// Exactly 1 after an abandon, however many scans the runner has left.
PROPERTY AbandonCalls : UDINT
GET
AbandonCalls := _AbandonCalls;
END_GET
END_PROPERTY

PROPERTY BodyCalls : UDINT
GET
BodyCalls := _BodyCalls;
END_GET
END_PROPERTY

METHOD Run : BOOL
VAR_INPUT
	Enable : BOOL;
	Test   : I_TestAssertions;
END_VAR
IF NOT Enable THEN
	_AbandonCalls := _AbandonCalls + 1;

	// Deliberately does NOT report itself finished. A test that hung will not

	// answer this either, and the runner must not wait for it.
	Run := FALSE;
	RETURN;
END_IF

_BodyCalls := _BodyCalls + 1;
Run		   := FALSE;
END_METHOD

// Always 0 - this double implements no teardown. Declared so a test can assert

// that abandonment did not somehow invent one.
PROPERTY TeardownCalls : UDINT
GET
TeardownCalls := 0;
END_GET
END_PROPERTY

END_FUNCTION_BLOCK

// ---- Tests/Runner/TEST_RunnerSetupDeadlineFires.TcPOU
// Setup has its OWN deadline. A fixture that never comes up must not run forever

// on the body's budget, and the body must never be reached.

//

// Teardown still runs: a fixture that half came up is exactly when cleanup

// matters.
FUNCTION_BLOCK TEST_RunnerSetupDeadlineFires IMPLEMENTS I_Test
VAR
	// A private runner, driven one scan per call. The outer test spans scans by

	// returning FALSE, which is exactly the mechanism being verified one level down.
	Registry	 : TestRegistry<1>;
	Runner		 : TestRunner;
	Handle		 : TestVerdict;
	Budgets		 : ST_TestBudgets;
	Journal		 : REFERENCE TO TestJournal;
	Slot		 : ST_TestSlot;
	Outcome		 : E_PhaseOutcome;
	Loaded		 : BOOL;
	Phase		 : DINT;
	Scans		 : DINT;
	Subject		 : HangingSetupTest;
	ExpectedZero : UDINT;
	ExpectedOne	 : UDINT;
	ExpectedTwo	 : UDINT;
	ActualCount	 : UDINT;
	ExpectedKind : E_FailureKind;
	ActualKind	 : E_FailureKind;
END_VAR

METHOD Run : BOOL
VAR_INPUT
	Enable : BOOL;
	Test   : I_TestAssertions;
END_VAR
Scans := Scans + 1;
IF Scans > 200 THEN
	Test.Fail('the subject never reached a terminal outcome');
	Run := TRUE;
	RETURN;
END_IF

CASE Phase OF
	0:
		Budgets.Setup.Cycles	  := 2;
		Budgets.Setup.IsCyclesSet := TRUE;

		// The body budget is deliberately left disabled. If the runner were using it

		// for setup, nothing would ever expire and the watchdog would fail this test.
		Registry.TryClaim(Subject, 'setup hangs', Budgets);
		Runner.Attach(Roster := Registry, Verdict := Handle);
		Slot   := Registry.Slot(0);
		Loaded := Runner.Load(Slot);
		Phase  := 1;
		Run	   := FALSE;

	1:
		Outcome := Runner.Advance(Enable := TRUE);
		IF Outcome <> E_PhaseOutcome.Running THEN
			Phase := 2;
		END_IF

		Run := FALSE;

	2:
		ExpectedTwo := 2;
		ActualCount := Subject.SetupCalls;
		Test.AssertEqual(ExpectedTwo, ActualCount, 'setup got its own budget, not the body one');
		ExpectedZero := 0;
		ActualCount	 := Subject.BodyCalls;
		Test.AssertEqual(ExpectedZero, ActualCount, 'the body was never reached');
		ExpectedOne := 1;
		ActualCount := Subject.TeardownCalls;
		Test.AssertEqual(ExpectedOne, ActualCount, 'teardown ran anyway');
		Journal REF= Registry.Journal(0);
		IF __ISVALIDREF(Journal) THEN
			ExpectedKind := E_FailureKind.Timeout;
			ActualKind	 := Journal.Kind;
			Test.AssertEqual(ExpectedKind, ActualKind, 'recorded as a timeout');
		END_IF

		Run := TRUE;
END_CASE
END_METHOD

END_FUNCTION_BLOCK

// ---- Doubles/HangingSetupTest.TcPOU
// Setup that never completes. Bounded by the SETUP deadline, not the body's - the

// body must never run, and teardown must still be called.
FUNCTION_BLOCK HangingSetupTest IMPLEMENTS I_Test, I_TestSetup, I_TestTeardown
VAR
	_SetupCalls	   : UDINT;
	_BodyCalls	   : UDINT;
	_TeardownCalls : UDINT;
END_VAR

// Must be 0. Setup never succeeded, so the body was never exercised.
PROPERTY BodyCalls : UDINT
GET
BodyCalls := _BodyCalls;
END_GET
END_PROPERTY

METHOD Run : BOOL
VAR_INPUT
	Enable : BOOL;
	Test   : I_TestAssertions;
END_VAR
IF Enable THEN
	_BodyCalls := _BodyCalls + 1;
END_IF

Run := TRUE;
END_METHOD

METHOD Setup : BOOL
VAR_INPUT
	Enable : BOOL;
	Test   : I_TestAssertions;
END_VAR
IF Enable THEN
	_SetupCalls := _SetupCalls + 1;
END_IF

Setup := FALSE;
END_METHOD

PROPERTY SetupCalls : UDINT
GET
SetupCalls := _SetupCalls;
END_GET
END_PROPERTY

METHOD Teardown : BOOL
VAR_INPUT
	Enable : BOOL;
	Test   : I_TestAssertions;
END_VAR
_TeardownCalls := _TeardownCalls + 1;
Teardown	   := TRUE;
END_METHOD

// Must be 1 even here. On a rig, a fixture that half came up is exactly when

// cleanup matters most.
PROPERTY TeardownCalls : UDINT
GET
TeardownCalls := _TeardownCalls;
END_GET
END_PROPERTY

END_FUNCTION_BLOCK

// ---- Tests/Runner/TEST_RunnerTeardownOverrunKeepsTheVerdict.TcPOU
// A passing test whose cleanup hangs still proved the code correct. The verdict

// stands.

//

// The overrun is reported separately - TeardownOverran, with a diagnostic and the

// label - because the SUITE has to raise a framework error for it and the runner

// holds no reporters. On a rig this may mean an axis left powered, so it must be

// loud without being a lie about the test.
FUNCTION_BLOCK TEST_RunnerTeardownOverrunKeepsTheVerdict IMPLEMENTS I_Test
VAR
	// A private runner, driven one scan per call. The outer test spans scans by

	// returning FALSE, which is exactly the mechanism being verified one level down.
	Registry	   : TestRegistry<1>;
	Runner		   : TestRunner;
	Handle		   : TestVerdict;
	Budgets		   : ST_TestBudgets;
	Journal		   : REFERENCE TO TestJournal;
	Slot		   : ST_TestSlot;
	Outcome		   : E_PhaseOutcome;
	Loaded		   : BOOL;
	Phase		   : DINT;
	Scans		   : DINT;
	Subject		   : HangingTeardownTest;
	ExpectedTwo	   : UDINT;
	ActualCount	   : UDINT;
	ExpectedStatus : E_TestStatus;
	ActualStatus   : E_TestStatus;
	Diagnostic	   : T_MaxString;
	ActiveLabel	   : T_MaxString;
	ExpectedLabel  : T_MaxString;
END_VAR

METHOD Run : BOOL
VAR_INPUT
	Enable : BOOL;
	Test   : I_TestAssertions;
END_VAR
Scans := Scans + 1;
IF Scans > 200 THEN
	Test.Fail('the subject never reached a terminal outcome');
	Run := TRUE;
	RETURN;
END_IF

CASE Phase OF
	0:
		Budgets.Teardown.Cycles		 := 2;
		Budgets.Teardown.IsCyclesSet := TRUE;
		Registry.TryClaim(Subject, 'teardown hangs', Budgets);
		Runner.Attach(Roster := Registry, Verdict := Handle);
		Slot   := Registry.Slot(0);
		Loaded := Runner.Load(Slot);
		Phase  := 1;
		Run	   := FALSE;

	1:
		Outcome := Runner.Advance(Enable := TRUE);
		IF Outcome <> E_PhaseOutcome.Running THEN
			// Read before anything else can unload it.
			Diagnostic	:= Runner.TeardownDiagnostic;
			ActiveLabel := Runner.ActiveLabel;
			Phase		:= 2;
		END_IF

		Run := FALSE;

	2:
		Test.AssertTrue(Outcome = E_PhaseOutcome.TeardownOverran, 'reported as an overrun');
		ExpectedTwo := 2;
		ActualCount := Subject.TeardownCalls;
		Test.AssertEqual(ExpectedTwo, ActualCount, 'teardown got its own budget');
		Test.AssertTrue(Diagnostic <> '', 'a diagnostic was composed');
		Test.AssertTrue(FIND(Diagnostic, 'teardown') > 0, 'and it names the phase');
		ExpectedLabel := 'teardown hangs';
		Test.AssertEqual(ExpectedLabel, ActiveLabel, 'and the test that hung');

		// The point of the whole test.
		Journal REF= Registry.Journal(0);
		IF __ISVALIDREF(Journal) THEN
			ExpectedStatus := E_TestStatus.Passed;
			ActualStatus   := Journal.Status;
			Test.AssertEqual(ExpectedStatus, ActualStatus, 'the verdict is untouched');
		END_IF

		Run := TRUE;
END_CASE
END_METHOD

END_FUNCTION_BLOCK

// ---- Doubles/HangingTeardownTest.TcPOU
// Passes cleanly, then hangs on the way out.

//

// The verdict must survive: a passing test whose cleanup hung still proved the

// code correct. The overrun is a framework error, not a test failure - but on a

// rig it may mean an axis left powered, so it must be loud.
FUNCTION_BLOCK HangingTeardownTest IMPLEMENTS I_Test, I_TestTeardown
VAR
	_BodyCalls	   : UDINT;
	_TeardownCalls : UDINT;
END_VAR

PROPERTY BodyCalls : UDINT
GET
BodyCalls := _BodyCalls;
END_GET
END_PROPERTY

METHOD Run : BOOL
VAR_INPUT
	Enable : BOOL;
	Test   : I_TestAssertions;
END_VAR
IF Enable THEN
	_BodyCalls := _BodyCalls + 1;
	Test.AssertTrue(TRUE, 'the body was fine');
END_IF

Run := TRUE;
END_METHOD

METHOD Teardown : BOOL
VAR_INPUT
	Enable : BOOL;
	Test   : I_TestAssertions;
END_VAR
IF Enable THEN
	_TeardownCalls := _TeardownCalls + 1;
END_IF

Teardown := FALSE;
END_METHOD

PROPERTY TeardownCalls : UDINT
GET
TeardownCalls := _TeardownCalls;
END_GET
END_PROPERTY

END_FUNCTION_BLOCK

// ---- Tests/Runner/TEST_RunnerAbandonMakesOneFinalCall.TcPOU
// Dropping Enable abandons the test. The phase in flight gets ONE final call so

// it can put its own state back, and the return is ignored - a test that hung will

// not answer that call either, and waiting for it would reproduce the stall the

// design removes.

//

// Teardown is NOT run. Abandonment is the suite being switched off, not a test

// finishing, and calling cleanup on a half-torn-down rig is its own hazard.
FUNCTION_BLOCK TEST_RunnerAbandonMakesOneFinalCall IMPLEMENTS I_Test
VAR
	// A private runner, driven one scan per call. The outer test spans scans by

	// returning FALSE, which is exactly the mechanism being verified one level down.
	Registry	   : TestRegistry<1>;
	Runner		   : TestRunner;
	Handle		   : TestVerdict;
	Budgets		   : ST_TestBudgets;
	Journal		   : REFERENCE TO TestJournal;
	Slot		   : ST_TestSlot;
	Outcome		   : E_PhaseOutcome;
	Loaded		   : BOOL;
	Phase		   : DINT;
	Scans		   : DINT;
	Subject		   : HangingBodyTest;
	ExpectedOne	   : UDINT;
	ExpectedZero   : UDINT;
	ActualCount	   : UDINT;
	ExpectedStatus : E_TestStatus;
	ActualStatus   : E_TestStatus;
END_VAR

METHOD Run : BOOL
VAR_INPUT
	Enable : BOOL;
	Test   : I_TestAssertions;
END_VAR
Scans := Scans + 1;
IF Scans > 200 THEN
	Test.Fail('the subject never reached a terminal outcome');
	Run := TRUE;
	RETURN;
END_IF

CASE Phase OF
	0:
		Registry.TryClaim(Subject, 'abandoned', Budgets);
		Runner.Attach(Roster := Registry, Verdict := Handle);
		Slot   := Registry.Slot(0);
		Loaded := Runner.Load(Slot);
		Phase  := 1;
		Run	   := FALSE;

	1:
		// Let it run a couple of scans first, so there is something to abandon.
		Outcome := Runner.Advance(Enable := TRUE);
		IF Subject.BodyCalls >= 2 THEN
			Phase := 2;
		END_IF

		Run := FALSE;

	2:
		Outcome := Runner.Advance(Enable := FALSE);
		Phase	:= 3;
		Run		:= FALSE;

	3:
		// A second abandon must not produce a second final call.
		Outcome := Runner.Advance(Enable := FALSE);
		Phase	:= 4;
		Run		:= FALSE;

	4:
		ExpectedOne := 1;
		ActualCount := Subject.AbandonCalls;
		Test.AssertEqual(ExpectedOne, ActualCount, 'exactly one call with Enable FALSE');
		ExpectedZero := 0;
		ActualCount	 := Subject.TeardownCalls;
		Test.AssertEqual(ExpectedZero, ActualCount, 'teardown was not run');
		Journal REF= Registry.Journal(0);
		IF __ISVALIDREF(Journal) THEN
			// Errored, not Failed: the code under test was never shown to be wrong. Not
			// Skipped either - an abandoned run must not read as a clean one.
			ExpectedStatus := E_TestStatus.Errored;
			ActualStatus   := Journal.Status;
			Test.AssertEqual(ExpectedStatus, ActualStatus, 'abandoned tests are Errored');
		END_IF

		Run := TRUE;
END_CASE
END_METHOD

END_FUNCTION_BLOCK

// ---- Tests/Runner/TEST_RunnerRefusesAnEmptySlot.TcPOU
// A slot carrying no test is refused, and nothing is loaded. A caller that has

// miscounted gets FALSE and an Idle runner rather than a dereferenced null.
FUNCTION_BLOCK TEST_RunnerRefusesAnEmptySlot IMPLEMENTS I_Test
VAR
	// A private runner, driven one scan per call. The outer test spans scans by

	// returning FALSE, which is exactly the mechanism being verified one level down.
	Registry  : TestRegistry<1>;
	Runner	  : TestRunner;
	Handle	  : TestVerdict;
	Budgets	  : ST_TestBudgets;
	Journal	  : REFERENCE TO TestJournal;
	Slot	  : ST_TestSlot;
	Outcome	  : E_PhaseOutcome;
	Loaded	  : BOOL;
	Phase	  : DINT;
	Scans	  : DINT;
	EmptySlot : ST_TestSlot;
	Refused	  : BOOL;
END_VAR

METHOD Run : BOOL
VAR_INPUT
	Enable : BOOL;
	Test   : I_TestAssertions;
END_VAR
Scans := Scans + 1;
IF Scans > 200 THEN
	Test.Fail('the subject never reached a terminal outcome');
	Run := TRUE;
	RETURN;
END_IF

Runner.Attach(Roster := Registry, Verdict := Handle);
Refused := Runner.Load(EmptySlot);
Test.AssertFalse(Refused, 'an empty slot is refused');
Test.AssertTrue(Runner.Outcome = E_PhaseOutcome.Idle, 'and nothing was loaded');

// Slot 0 of an empty registry is also empty - the registry hands back a defined

// empty slot rather than whatever was nearby.
Slot	:= Registry.Slot(0);
Refused := Runner.Load(Slot);
Test.AssertFalse(Refused, 'an unregistered index is refused too');
Test.AssertTrue(Runner.Outcome = E_PhaseOutcome.Idle, 'still nothing loaded');
Run := TRUE;
END_METHOD

END_FUNCTION_BLOCK

// ---- Tests/Suite/TEST_SuiteRunsEveryRegisteredTest.TcPOU
// The whole loop: register three, drive to completion, and every one of them ran

// exactly once and was counted.
FUNCTION_BLOCK TEST_SuiteRunsEveryRegisteredTest IMPLEMENTS I_Test
VAR
	// A private suite, driven one scan per call. The outer test spans scans by

	// returning FALSE - which is the mechanism the inner suite is being asked to

	// drive, one level down.
	Inner			: TestSuite<4>;
	Budgets			: ST_TestBudgets;
	Phase			: DINT;
	Scans			: DINT;
	A				: PassingTest;
	B				: PassingTest;
	C				: PassingTest;
	ExpectedCount	: UDINT;
	ActualCount		: UDINT;
	ExpectedOutcome : E_RunOutcome;
	ActualOutcome	: E_RunOutcome;
END_VAR

METHOD Run : BOOL
VAR_INPUT
	Enable : BOOL;
	Test   : I_TestAssertions;
END_VAR
Scans := Scans + 1;
IF Scans > 200 THEN
	Test.Fail('the inner suite never completed');
	Run := TRUE;
	RETURN;
END_IF

CASE Phase OF
	0:
		Inner.SetLabel('inner');
		Inner.Register(A, 'first', Budgets);
		Inner.Register(B, 'second', Budgets);
		Inner.Register(C, 'third', Budgets);
		Phase := 1;
		Run	  := FALSE;

	1:
		IF Inner.Run(Enable := TRUE) THEN
			Phase := 2;
		END_IF

		Run := FALSE;

	2:
		Test.AssertTrue(Inner.IsComplete, 'the run finished');
		ExpectedCount := 3;
		ActualCount	  := Inner.TestCount;
		Test.AssertEqual(ExpectedCount, ActualCount, 'three registered');
		ActualCount := Inner.PassedCount;
		Test.AssertEqual(ExpectedCount, ActualCount, 'three passed');
		ExpectedCount := 0;
		ActualCount	  := Inner.FailedCount;
		Test.AssertEqual(ExpectedCount, ActualCount, 'none failed');
		ExpectedCount := 1;
		ActualCount	  := A.BodyCalls;
		Test.AssertEqual(ExpectedCount, ActualCount, 'the first ran once');
		ActualCount := C.BodyCalls;
		Test.AssertEqual(ExpectedCount, ActualCount, 'and so did the last');
		ExpectedOutcome := E_RunOutcome.Passed;
		ActualOutcome	:= Inner.Outcome;
		Test.AssertEqual(ExpectedOutcome, ActualOutcome, 'the run passed');
		Run := TRUE;
END_CASE
END_METHOD

END_FUNCTION_BLOCK

// ---- Doubles/PassingTest.TcPOU
// Passes in one scan. The baseline for suite-level counting.

//

// Records a check deliberately: a body that checks nothing is reported Errored,

// not Passed, so a double that asserted nothing would quietly test the wrong

// thing.
FUNCTION_BLOCK PassingTest IMPLEMENTS I_Test
VAR
	_BodyCalls : UDINT;
END_VAR

// How many times a suite has run this. A re-run doubles it; an individual re-run

// raises it without touching any count the suite reports.
PROPERTY BodyCalls : UDINT
GET
BodyCalls := _BodyCalls;
END_GET
END_PROPERTY

METHOD Run : BOOL
VAR_INPUT
	Enable : BOOL;
	Test   : I_TestAssertions;
END_VAR
IF NOT Enable THEN
	Run := TRUE;
	RETURN;
END_IF

_BodyCalls := _BodyCalls + 1;
Test.AssertTrue(TRUE, 'this one passes');
Run := TRUE;
END_METHOD

END_FUNCTION_BLOCK

// ---- Tests/Suite/TEST_SuiteSeparatesFailuresFromErrors.TcPOU
// Failed and Errored are different signals and are counted apart.

//

// A failure means the code is wrong. An error means the run cannot be trusted -

// and Errored outranks Failed in the aggregate, because a framework or environment

// problem casts doubt on every other result.
FUNCTION_BLOCK TEST_SuiteSeparatesFailuresFromErrors IMPLEMENTS I_Test
VAR
	// A private suite, driven one scan per call. The outer test spans scans by

	// returning FALSE - which is the mechanism the inner suite is being asked to

	// drive, one level down.
	Inner			: TestSuite<4>;
	Budgets			: ST_TestBudgets;
	Phase			: DINT;
	Scans			: DINT;
	Good			: PassingTest;
	Bad				: FailingTest;
	Ugly			: ErroringTest;
	ExpectedCount	: UDINT;
	ActualCount		: UDINT;
	ExpectedOutcome : E_RunOutcome;
	ActualOutcome	: E_RunOutcome;
END_VAR

METHOD Run : BOOL
VAR_INPUT
	Enable : BOOL;
	Test   : I_TestAssertions;
END_VAR
Scans := Scans + 1;
IF Scans > 200 THEN
	Test.Fail('the inner suite never completed');
	Run := TRUE;
	RETURN;
END_IF

CASE Phase OF
	0:
		Inner.SetLabel('inner');
		Inner.Register(Good, 'passes', Budgets);
		Inner.Register(Bad, 'fails', Budgets);
		Inner.Register(Ugly, 'errors', Budgets);
		Phase := 1;
		Run	  := FALSE;

	1:
		IF Inner.Run(Enable := TRUE) THEN
			Phase := 2;
		END_IF

		Run := FALSE;

	2:
		ExpectedCount := 1;
		ActualCount	  := Inner.PassedCount;
		Test.AssertEqual(ExpectedCount, ActualCount, 'one passed');
		ActualCount := Inner.FailedCount;
		Test.AssertEqual(ExpectedCount, ActualCount, 'one failed');
		ActualCount := Inner.ErrorCount;
		Test.AssertEqual(ExpectedCount, ActualCount, 'one errored');
		ExpectedCount := 3;
		ActualCount	  := Inner.TestCount;
		Test.AssertEqual(ExpectedCount, ActualCount, 'and they add up to the registered count');

		// Errored outranks Failed.
		ExpectedOutcome := E_RunOutcome.Errored;
		ActualOutcome	:= Inner.Outcome;
		Test.AssertEqual(ExpectedOutcome, ActualOutcome, 'an error outranks a failure');
		Run := TRUE;
END_CASE
END_METHOD

END_FUNCTION_BLOCK

// ---- Doubles/FailingTest.TcPOU
// Fails in one scan, on purpose. Proves FailedCount moves and that a failure

// carries the run's outcome with it.
FUNCTION_BLOCK FailingTest IMPLEMENTS I_Test
VAR
	_BodyCalls : UDINT;
END_VAR

// How many times a suite has run this. A re-run doubles it; an individual re-run

// raises it without touching any count the suite reports.
PROPERTY BodyCalls : UDINT
GET
BodyCalls := _BodyCalls;
END_GET
END_PROPERTY

METHOD Run : BOOL
VAR_INPUT
	Enable : BOOL;
	Test   : I_TestAssertions;
END_VAR
IF NOT Enable THEN
	Run := TRUE;
	RETURN;
END_IF

_BodyCalls := _BodyCalls + 1;
Test.Fail('this one fails, deliberately');
Run := TRUE;
END_METHOD

END_FUNCTION_BLOCK

// ---- Doubles/ErroringTest.TcPOU
// Reports an environmental problem rather than a failure. The code under test was

// never exercised, so the run cannot be trusted - which is a different signal from

// the code being wrong, and must be counted separately.
FUNCTION_BLOCK ErroringTest IMPLEMENTS I_Test
VAR
	_BodyCalls : UDINT;
END_VAR

// How many times a suite has run this. A re-run doubles it; an individual re-run

// raises it without touching any count the suite reports.
PROPERTY BodyCalls : UDINT
GET
BodyCalls := _BodyCalls;
END_GET
END_PROPERTY

METHOD Run : BOOL
VAR_INPUT
	Enable : BOOL;
	Test   : I_TestAssertions;
END_VAR
IF NOT Enable THEN
	Run := TRUE;
	RETURN;
END_IF

_BodyCalls := _BodyCalls + 1;
Test.ReportError('the fixture was not available');
Run := TRUE;
END_METHOD

END_FUNCTION_BLOCK

// ---- Tests/Suite/TEST_SuiteClosesRegistrationOnFirstEnable.TcPOU
// Registration is open until the suite is first enabled, and not after. A late

// registration is refused AND reported - a test that vanished silently would leave

// CI seeing fewer passes rather than a failure.
FUNCTION_BLOCK TEST_SuiteClosesRegistrationOnFirstEnable IMPLEMENTS I_Test
VAR
	// A private suite, driven one scan per call. The outer test spans scans by

	// returning FALSE - which is the mechanism the inner suite is being asked to

	// drive, one level down.
	Inner		  : TestSuite<4>;
	Budgets		  : ST_TestBudgets;
	Phase		  : DINT;
	Scans		  : DINT;
	Early		  : PassingTest;
	Late		  : PassingTest;
	AcceptedEarly : BOOL;
	AcceptedLate  : BOOL;
	OpenAtStart	  : BOOL;
	OpenAfter	  : BOOL;
	ExpectedCount : UDINT;
	ActualCount	  : UDINT;
END_VAR

METHOD Run : BOOL
VAR_INPUT
	Enable : BOOL;
	Test   : I_TestAssertions;
END_VAR
Scans := Scans + 1;
IF Scans > 200 THEN
	Test.Fail('the inner suite never completed');
	Run := TRUE;
	RETURN;
END_IF

CASE Phase OF
	0:
		Inner.SetLabel('inner');
		OpenAtStart	  := Inner.IsOpen;
		AcceptedEarly := Inner.Register(Early, 'in time', Budgets);
		Phase		  := 1;
		Run			  := FALSE;

	1:
		// One scan of the suite closes the window.
		Inner.Run(Enable := TRUE);
		OpenAfter	 := Inner.IsOpen;
		AcceptedLate := Inner.Register(Late, 'too late', Budgets);
		Phase		 := 2;
		Run			 := FALSE;

	2:
		IF Inner.Run(Enable := TRUE) THEN
			Phase := 3;
		END_IF

		Run := FALSE;

	3:
		Test.AssertTrue(OpenAtStart, 'open before the first enable');
		Test.AssertTrue(AcceptedEarly, 'the early registration was taken');
		Test.AssertFalse(OpenAfter, 'closed once enabled');
		Test.AssertFalse(AcceptedLate, 'the late one was refused');
		ExpectedCount := 1;
		ActualCount	  := Inner.TestCount;
		Test.AssertEqual(ExpectedCount, ActualCount, 'and took no slot');
		ExpectedCount := 0;
		ActualCount	  := Late.BodyCalls;
		Test.AssertEqual(ExpectedCount, ActualCount, 'the late test never ran');

		// Refused, and said so.
		Test.AssertTrue(Inner.ErrorCount > 0, 'the rejection was reported, not silent');
		Run := TRUE;
END_CASE
END_METHOD

END_FUNCTION_BLOCK

// ---- Tests/Suite/TEST_SuiteRejectedRegistrationIsNeverSilent.TcPOU
// A duplicate label is refused and raises a framework error. Labels are the key

// CI trend history is built on, so two tests cannot share one - and a test that

// failed to register must not simply disappear.
FUNCTION_BLOCK TEST_SuiteRejectedRegistrationIsNeverSilent IMPLEMENTS I_Test
VAR
	// A private suite, driven one scan per call. The outer test spans scans by

	// returning FALSE - which is the mechanism the inner suite is being asked to

	// drive, one level down.
	Inner			: TestSuite<4>;
	Budgets			: ST_TestBudgets;
	Phase			: DINT;
	Scans			: DINT;
	First			: PassingTest;
	Second			: PassingTest;
	AcceptedFirst	: BOOL;
	AcceptedSecond	: BOOL;
	ExpectedCount	: UDINT;
	ActualCount		: UDINT;
	ExpectedOutcome : E_RunOutcome;
	ActualOutcome	: E_RunOutcome;
END_VAR

METHOD Run : BOOL
VAR_INPUT
	Enable : BOOL;
	Test   : I_TestAssertions;
END_VAR
Scans := Scans + 1;
IF Scans > 200 THEN
	Test.Fail('the inner suite never completed');
	Run := TRUE;
	RETURN;
END_IF

CASE Phase OF
	0:
		Inner.SetLabel('inner');
		AcceptedFirst  := Inner.Register(First, 'same label', Budgets);
		AcceptedSecond := Inner.Register(Second, 'same label', Budgets);
		Phase		   := 1;
		Run			   := FALSE;

	1:
		IF Inner.Run(Enable := TRUE) THEN
			Phase := 2;
		END_IF

		Run := FALSE;

	2:
		Test.AssertTrue(AcceptedFirst, 'the first was taken');
		Test.AssertFalse(AcceptedSecond, 'the duplicate was refused');
		ExpectedCount := 1;
		ActualCount	  := Inner.TestCount;
		Test.AssertEqual(ExpectedCount, ActualCount, 'only one slot used');
		Test.AssertTrue(Inner.ErrorCount > 0, 'the rejection reached the counts');

		// A rejection raised BEFORE the run must survive Tally.Begin, or the run goes

		// green while a test is missing from it.
		ExpectedOutcome := E_RunOutcome.Errored;
		ActualOutcome	:= Inner.Outcome;
		Test.AssertEqual(ExpectedOutcome, ActualOutcome, 'and turned the run red');
		Run := TRUE;
END_CASE
END_METHOD

END_FUNCTION_BLOCK

// ---- Tests/Suite/TEST_SuiteSkipMarksEverythingSkipped.TcPOU
// A skipped suite is COMPLETE, not stuck. If it reported otherwise, any sequencer

// aggregating it would wait for it forever.

//

// No body runs, nothing is a failure, and Skip closes the registration window -

// the suite has reached a terminal state, so registration cannot reopen.
FUNCTION_BLOCK TEST_SuiteSkipMarksEverythingSkipped IMPLEMENTS I_Test
VAR
	// A private suite, driven one scan per call. The outer test spans scans by

	// returning FALSE - which is the mechanism the inner suite is being asked to

	// drive, one level down.
	Inner			: TestSuite<4>;
	Budgets			: ST_TestBudgets;
	Phase			: DINT;
	Scans			: DINT;
	A				: PassingTest;
	B				: FailingTest;
	ExpectedCount	: UDINT;
	ActualCount		: UDINT;
	ExpectedOutcome : E_RunOutcome;
	ActualOutcome	: E_RunOutcome;
END_VAR

METHOD Run : BOOL
VAR_INPUT
	Enable : BOOL;
	Test   : I_TestAssertions;
END_VAR
Scans := Scans + 1;
IF Scans > 200 THEN
	Test.Fail('the inner suite never completed');
	Run := TRUE;
	RETURN;
END_IF

CASE Phase OF
	0:
		Inner.SetLabel('inner');
		Inner.Register(A, 'would pass', Budgets);
		Inner.Register(B, 'would fail', Budgets);
		Inner.Skip();
		Phase := 1;
		Run	  := FALSE;

	1:
		// Complete already; Run must not restart anything.
		Inner.Run(Enable := TRUE);
		Phase := 2;
		Run	  := FALSE;

	2:
		Test.AssertTrue(Inner.IsComplete, 'a skipped suite is complete');
		Test.AssertFalse(Inner.IsOpen, 'and registration is closed');
		ExpectedCount := 2;
		ActualCount	  := Inner.SkippedCount;
		Test.AssertEqual(ExpectedCount, ActualCount, 'both are skipped');
		ExpectedCount := 0;
		ActualCount	  := Inner.FailedCount;
		Test.AssertEqual(ExpectedCount, ActualCount, 'nothing failed');

		// The one that WOULD have failed never ran.
		ActualCount := B.BodyCalls;
		Test.AssertEqual(ExpectedCount, ActualCount, 'no body was called');
		ActualCount := A.BodyCalls;
		Test.AssertEqual(ExpectedCount, ActualCount, 'not even the passing one');

		// Skipped must not turn a build red.
		ExpectedOutcome := E_RunOutcome.Skipped;
		ActualOutcome	:= Inner.Outcome;
		Test.AssertEqual(ExpectedOutcome, ActualOutcome, 'the outcome is Skipped');
		Run := TRUE;
END_CASE
END_METHOD

END_FUNCTION_BLOCK

// ---- Tests/Suite/TEST_SuiteSkippedAfterARejectedRegistrationIsErrored.TcPOU
// A registration refused before a suite was skipped is still counted: the suite
// is Errored, not Skipped.
//
// The skipped twin of TEST_SuiteRejectedRegistrationIsNeverSilent, whose point is
// that a rejection raised before the run must survive Tally.Begin. StartRun
// re-applies it. Skip also calls Tally.Begin, and once re-applied nothing - so a
// wiring error in a skipped suite vanished from the counts, and the run stayed
// clear of red while a test was missing from it.
//
// A wiring error outranks a skip. The skip is still honoured: the test that did
// register is skipped, and never runs.
FUNCTION_BLOCK TEST_SuiteSkippedAfterARejectedRegistrationIsErrored IMPLEMENTS I_Test
VAR
	Inner			: TestSuite<4>;

	First			: PassingTest;
	Second			: PassingTest;
	AcceptedFirst	: BOOL;
	AcceptedSecond	: BOOL;

	Budgets : ST_TestBudgets;
	Phase	: DINT;
	Scans	: DINT;

	ExpectedCount : UDINT;
	ActualCount	  : UDINT;
	ExpectedOutcome : E_RunOutcome;
	ActualOutcome	: E_RunOutcome;
END_VAR

METHOD Run : BOOL
VAR_INPUT
	Enable : BOOL;
	Test   : I_TestAssertions;
END_VAR
Scans := Scans + 1;
IF Scans > 200 THEN
	Test.Fail('the inner suite never completed');
	Run := TRUE;
	RETURN;
END_IF

CASE Phase OF

0:
	Inner.SetLabel('inner');
	AcceptedFirst  := Inner.Register(First, 'same label', Budgets);
	AcceptedSecond := Inner.Register(Second, 'same label', Budgets);
	Inner.Skip();
	Phase := 1;
	Run	  := FALSE;

1:
	IF Inner.Run(Enable := TRUE) THEN
		Phase := 2;
	END_IF
	Run := FALSE;

2:
	Test.AssertTrue(AcceptedFirst, 'the first was taken');
	Test.AssertFalse(AcceptedSecond, 'the duplicate was refused');

	ExpectedCount := 1;
	ActualCount	  := Inner.ErrorCount;
	Test.AssertEqual(ExpectedCount, ActualCount, 'the refusal survived the skip, counted once');

	ActualCount := Inner.SkippedCount;
	Test.AssertEqual(ExpectedCount, ActualCount, 'the test that registered was skipped');
	ExpectedCount := 0;
	ActualCount	  := First.BodyCalls;
	Test.AssertEqual(ExpectedCount, ActualCount, 'and never ran');

	ExpectedOutcome := E_RunOutcome.Errored;
	ActualOutcome	:= Inner.Outcome;
	Test.AssertEqual(ExpectedOutcome, ActualOutcome, 'a wiring error outranks the skip');

	Run := TRUE;

END_CASE
END_METHOD

END_FUNCTION_BLOCK

// ---- Tests/Suite/TEST_SuiteSkippedWithNoLabelIsAFrameworkError.TcPOU
// A skipped suite with no label is a framework error, as an enabled one is.
//
// The skipped twin of TEST_SuiteWithNoLabelIsAFrameworkError. An unnamed suite
// produces an unnamed node in the result document, which no CI system can group
// by, and StartRun reports it. Skip never passes through StartRun, so an unnamed
// skipped suite went into the document without a word.
//
// The sink is attached before the skip so the error is not only counted but SAID:
// a count with no reason behind it sends a reader looking in the wrong place.
FUNCTION_BLOCK TEST_SuiteSkippedWithNoLabelIsAFrameworkError IMPLEMENTS I_Test
VAR
	Inner	: TestSuite<4>;
	Spy		: SpyReporter;
	A		: PassingTest;

	Budgets : ST_TestBudgets;
	Phase	: DINT;
	Scans	: DINT;

	ExpectedCount : UDINT;
	ActualCount	  : UDINT;
	ExpectedOutcome : E_RunOutcome;
	ActualOutcome	: E_RunOutcome;
END_VAR

METHOD Run : BOOL
VAR_INPUT
	Enable : BOOL;
	Test   : I_TestAssertions;
END_VAR
Scans := Scans + 1;
IF Scans > 200 THEN
	Test.Fail('the inner suite never completed');
	Run := TRUE;
	RETURN;
END_IF

CASE Phase OF

0:
	// Deliberately no SetLabel.
	Inner.Register(A, 'a test', Budgets);
	Inner.AddReporter(Spy);
	Inner.Skip();
	Phase := 1;
	Run	  := FALSE;

1:
	IF Inner.Run(Enable := TRUE) THEN
		Phase := 2;
	END_IF
	Run := FALSE;

2:
	ExpectedCount := 1;
	ActualCount	  := Inner.ErrorCount;
	Test.AssertEqual(ExpectedCount, ActualCount, 'the missing label was counted');
	ActualCount := Spy.FrameworkErrorCalls;
	Test.AssertEqual(ExpectedCount, ActualCount, 'and said, to the sink attached before the skip');

	ActualCount := Inner.SkippedCount;
	Test.AssertEqual(ExpectedCount, ActualCount, 'the test was still skipped');
	ExpectedCount := 0;
	ActualCount	  := A.BodyCalls;
	Test.AssertEqual(ExpectedCount, ActualCount, 'and never ran');

	ExpectedOutcome := E_RunOutcome.Errored;
	ActualOutcome	:= Inner.Outcome;
	Test.AssertEqual(ExpectedOutcome, ActualOutcome, 'the suite is Errored, not quietly Skipped');

	Run := TRUE;

END_CASE
END_METHOD

END_FUNCTION_BLOCK

// ---- Doubles/SpyReporter.TcPOU
// A reporter that records what it was told, and nothing else.

//

// Implements BOTH faces: I_TestReporter for verdicts, I_TestDetailSink for

// individual checks. VerdictOnlyReporter is the counterpart that implements only

// the first, and the pair together are what proves the fan-out asks each sink what

// it actually wants rather than calling everything on everyone.
FUNCTION_BLOCK SpyReporter IMPLEMENTS I_TestReporter, I_TestDetailSink
VAR
	_CyclicCalls		   : UDINT;
	_TestFinishedCalls	   : UDINT;
	_SuiteFinishedCalls	   : UDINT;
	_RunFinishedCalls	   : UDINT;
	_RunStartedCalls	   : UDINT;
	_StartedBeforeAnything : BOOL;
	_FrameworkErrorCalls   : UDINT;
	_TestStartedCalls	   : UDINT;
	_CheckCalls			   : UDINT;
	_CheckPassedCalls	   : UDINT;
	_CheckFailedCalls	   : UDINT;
	_LastTestLabel		   : T_MaxString;
	_LastSuiteLabel		   : T_MaxString;
	_LastSummary		   : T_MaxString;
	_LastExpected		   : T_MaxString;
	_LastActual			   : T_MaxString;
	_LastErrorSource	   : T_MaxString;
	_LastErrorMessage	   : T_MaxString;
	_LastStatus			   : E_TestStatus;
	_LastSuiteOutcome	   : E_RunOutcome;
	_LastSuitePassed	   : UDINT;
	_StartedBeforeChecks   : BOOL;
	_IsBusy				   : BOOL;
	_Ordinal			   : UDINT;
	_Witness			   : I_ProbeWitness;
END_VAR

PROPERTY CheckCalls : UDINT
GET
CheckCalls := _CheckCalls;
END_GET
END_PROPERTY

METHOD CheckFailed
VAR_INPUT
	StepLabel  : T_MaxString;
	Kind	   : E_FailureKind;
	Expected   : T_MaxString;
	Actual	   : T_MaxString;
	Diagnostic : T_MaxString;
	Message	   : T_MaxString;
END_VAR
_CheckCalls		  := _CheckCalls + 1;
_CheckFailedCalls := _CheckFailedCalls + 1;
_LastExpected	  := Expected;
_LastActual		  := Actual;
END_METHOD

PROPERTY CheckFailedCalls : UDINT
GET
CheckFailedCalls := _CheckFailedCalls;
END_GET
END_PROPERTY

METHOD CheckPassed
VAR_INPUT
	StepLabel : T_MaxString;
	Detail	  : T_MaxString;
END_VAR
_CheckCalls		  := _CheckCalls + 1;
_CheckPassedCalls := _CheckPassedCalls + 1;
END_METHOD

PROPERTY CheckPassedCalls : UDINT
GET
CheckPassedCalls := _CheckPassedCalls;
END_GET
END_PROPERTY

// Identify this spy and give it somewhere to record the order it was called in.
METHOD Configure
VAR_INPUT
	Ordinal : UDINT;
	Witness : I_ProbeWitness;
END_VAR
_Ordinal := Ordinal;
_Witness := Witness;
END_METHOD

PROPERTY CyclicCalls : UDINT
GET
CyclicCalls := _CyclicCalls;
END_GET
END_PROPERTY

METHOD CyclicLogic
_CyclicCalls := _CyclicCalls + 1;
END_METHOD

METHOD FrameworkError
VAR_INPUT
	Source	: T_MaxString;
	Message : T_MaxString;
END_VAR
_FrameworkErrorCalls := _FrameworkErrorCalls + 1;
_LastErrorSource	 := Source;
_LastErrorMessage	 := Message;
END_METHOD

PROPERTY FrameworkErrorCalls : UDINT
GET
FrameworkErrorCalls := _FrameworkErrorCalls;
END_GET
END_PROPERTY

// FALSE while this spy claims work in flight. The fan-out ANDs every sink.
PROPERTY IsIdle : BOOL
GET
IsIdle := NOT _IsBusy;
END_GET
END_PROPERTY

PROPERTY LastActual : T_MaxString
GET
LastActual := _LastActual;
END_GET
END_PROPERTY

PROPERTY LastErrorMessage : T_MaxString
GET
LastErrorMessage := _LastErrorMessage;
END_GET
END_PROPERTY

PROPERTY LastErrorSource : T_MaxString
GET
LastErrorSource := _LastErrorSource;
END_GET
END_PROPERTY

PROPERTY LastExpected : T_MaxString
GET
LastExpected := _LastExpected;
END_GET
END_PROPERTY

PROPERTY LastStatus : E_TestStatus
GET
LastStatus := _LastStatus;
END_GET
END_PROPERTY

PROPERTY LastSuiteLabel : T_MaxString
GET
LastSuiteLabel := _LastSuiteLabel;
END_GET
END_PROPERTY

PROPERTY LastSuiteOutcome : E_RunOutcome
GET
LastSuiteOutcome := _LastSuiteOutcome;
END_GET
END_PROPERTY

PROPERTY LastSuitePassed : UDINT
GET
LastSuitePassed := _LastSuitePassed;
END_GET
END_PROPERTY

PROPERTY LastSummary : T_MaxString
GET
LastSummary := _LastSummary;
END_GET
END_PROPERTY

PROPERTY LastTestLabel : T_MaxString
GET
LastTestLabel := _LastTestLabel;
END_GET
END_PROPERTY

METHOD RunFinished
VAR_INPUT
	Status	   : I_TestRunStatus;
	TargetInfo : T_MaxString;
END_VAR
_RunFinishedCalls := _RunFinishedCalls + 1;
END_METHOD

PROPERTY RunFinishedCalls : UDINT
GET
RunFinishedCalls := _RunFinishedCalls;
END_GET
END_PROPERTY

// Counted, and the label kept - so a test can prove the run announced itself

// BEFORE anything else in it arrived, which is the whole point of the call.
METHOD RunStarted
VAR_INPUT
	Label	   : T_MaxString;
	TargetInfo : T_MaxString;
END_VAR
_RunStartedCalls	   := _RunStartedCalls + 1;
_StartedBeforeAnything := (_TestFinishedCalls = 0) AND (_SuiteFinishedCalls = 0);
END_METHOD

PROPERTY RunStartedCalls : UDINT
GET
RunStartedCalls := _RunStartedCalls;
END_GET
END_PROPERTY

// Pretend to have asynchronous work in flight, so IsIdle can be checked without a

// real file write.
METHOD SetBusy
VAR_INPUT
	Busy : BOOL;
END_VAR
_IsBusy := Busy;
END_METHOD

// TRUE if RunStarted arrived before any test or suite result. The ordering IS the

// contract - a sink that opens a document on this call has nowhere to put a result

// that arrived first.
PROPERTY StartedBeforeAnything : BOOL
GET
StartedBeforeAnything := _StartedBeforeAnything;
END_GET
END_PROPERTY

// TRUE if TestStarted arrived before any check did. The ordering guarantee is the

// whole reason TestStarted exists - a sink building a document has nowhere to put

// a check until it has been told to open an element.
PROPERTY StartedBeforeChecks : BOOL
GET
StartedBeforeChecks := _StartedBeforeChecks;
END_GET
END_PROPERTY

METHOD SuiteFinished
VAR_INPUT
	Status : I_TestRunStatus;
END_VAR
_SuiteFinishedCalls := _SuiteFinishedCalls + 1;
IF Status <> 0 THEN
	_LastSuiteOutcome := Status.Outcome;
	_LastSuitePassed  := Status.PassedCount;
END_IF
END_METHOD

PROPERTY SuiteFinishedCalls : UDINT
GET
SuiteFinishedCalls := _SuiteFinishedCalls;
END_GET
END_PROPERTY

METHOD TestFinished
VAR_INPUT
	SuiteLabel	  : T_MaxString;
	TestLabel	  : T_MaxString;
	Location	  : T_MaxString;
	Status		  : E_TestStatus;
	Kind		  : E_FailureKind;
	Summary		  : T_MaxString;
	ElapsedTime	  : LREAL;
	ElapsedCycles : UDINT;
	Assertions	  : UDINT;
END_VAR
_TestFinishedCalls := _TestFinishedCalls + 1;
_LastTestLabel	   := TestLabel;
_LastSuiteLabel	   := SuiteLabel;
_LastStatus		   := Status;
_LastSummary	   := Summary;
// Order of notification is order of attachment. Each spy stamps itself into a

// shared witness so a test can read the sequence back.
IF _Witness <> 0 THEN
	_Witness.Note(_Ordinal);
END_IF
END_METHOD

PROPERTY TestFinishedCalls : UDINT
GET
TestFinishedCalls := _TestFinishedCalls;
END_GET
END_PROPERTY

METHOD TestStarted
VAR_INPUT
	SuiteLabel : T_MaxString;
	TestLabel  : T_MaxString;
	Location   : T_MaxString;
END_VAR
_TestStartedCalls	 := _TestStartedCalls + 1;
_StartedBeforeChecks := (_CheckCalls = 0);
END_METHOD

PROPERTY TestStartedCalls : UDINT
GET
TestStartedCalls := _TestStartedCalls;
END_GET
END_PROPERTY

END_FUNCTION_BLOCK

// ---- Tests/Suite/TEST_SuiteReRunRepeatsTheRegisteredSet.TcPOU
// A re-run re-executes what was registered; it does not redefine it. The counts

// start again from nothing, every body runs a second time, and the window stays

// shut.
FUNCTION_BLOCK TEST_SuiteReRunRepeatsTheRegisteredSet IMPLEMENTS I_Test
VAR
	// A private suite, driven one scan per call. The outer test spans scans by

	// returning FALSE - which is the mechanism the inner suite is being asked to

	// drive, one level down.
	Inner		  : TestSuite<4>;
	Budgets		  : ST_TestBudgets;
	Phase		  : DINT;
	Scans		  : DINT;
	A			  : PassingTest;
	B			  : PassingTest;
	ExpectedCount : UDINT;
	ActualCount	  : UDINT;
END_VAR

METHOD Run : BOOL
VAR_INPUT
	Enable : BOOL;
	Test   : I_TestAssertions;
END_VAR
Scans := Scans + 1;
IF Scans > 200 THEN
	Test.Fail('the inner suite never completed');
	Run := TRUE;
	RETURN;
END_IF

CASE Phase OF
	0:
		Inner.SetLabel('inner');
		Inner.Register(A, 'first', Budgets);
		Inner.Register(B, 'second', Budgets);
		Phase := 1;
		Run	  := FALSE;

	1:
		IF Inner.Run(Enable := TRUE) THEN
			Phase := 2;
		END_IF

		Run := FALSE;

	2:
		ExpectedCount := 2;
		ActualCount	  := Inner.PassedCount;
		Test.AssertEqual(ExpectedCount, ActualCount, 'the first run passed both');
		Inner.ReRun();
		Test.AssertFalse(Inner.IsComplete, 'a re-run clears completion');
		Test.AssertFalse(Inner.IsOpen, 'and does not reopen registration');
		Phase := 3;
		Run	  := FALSE;

	3:
		IF Inner.Run(Enable := TRUE) THEN
			Phase := 4;
		END_IF

		Run := FALSE;

	4:
		ExpectedCount := 2;
		ActualCount	  := Inner.PassedCount;
		Test.AssertEqual(ExpectedCount, ActualCount, 'the counts started again, not doubled');
		ActualCount := Inner.TestCount;
		Test.AssertEqual(ExpectedCount, ActualCount, 'the registered set is unchanged');

		// The bodies, however, really did run twice.
		ActualCount := A.BodyCalls;
		Test.AssertEqual(ExpectedCount, ActualCount, 'the first test ran twice');
		ActualCount := B.BodyCalls;
		Test.AssertEqual(ExpectedCount, ActualCount, 'and so did the second');
		Run := TRUE;
END_CASE
END_METHOD

END_FUNCTION_BLOCK

// ---- Tests/Suite/TEST_SuiteReRunSingleRecordsNothing.TcPOU
// Re-running one test is a debugging aid, not a result. It really runs the test -

// otherwise it would be useless - and records NOTHING: no count moves, and with

// reporters attached nothing would reach them either.

//

// Without that, a session at the keyboard would pollute the CI artifact with

// duplicate entries.
FUNCTION_BLOCK TEST_SuiteReRunSingleRecordsNothing IMPLEMENTS I_Test
VAR
	// A private suite, driven one scan per call. The outer test spans scans by

	// returning FALSE - which is the mechanism the inner suite is being asked to

	// drive, one level down.
	Inner		  : TestSuite<4>;
	Budgets		  : ST_TestBudgets;
	Phase		  : DINT;
	Scans		  : DINT;
	A			  : PassingTest;
	B			  : PassingTest;
	Accepted	  : BOOL;
	Unknown		  : BOOL;
	PassedBefore  : UDINT;
	ExpectedCount : UDINT;
	ActualCount	  : UDINT;
END_VAR

METHOD Run : BOOL
VAR_INPUT
	Enable : BOOL;
	Test   : I_TestAssertions;
END_VAR
Scans := Scans + 1;
IF Scans > 200 THEN
	Test.Fail('the inner suite never completed');
	Run := TRUE;
	RETURN;
END_IF

CASE Phase OF
	0:
		Inner.SetLabel('inner');
		Inner.Register(A, 'first', Budgets);
		Inner.Register(B, 'second', Budgets);
		Phase := 1;
		Run	  := FALSE;

	1:
		IF Inner.Run(Enable := TRUE) THEN
			PassedBefore := Inner.PassedCount;
			Phase		 := 2;
		END_IF

		Run := FALSE;

	2:
		Unknown	 := Inner.ReRunSingle('no such label');
		Accepted := Inner.ReRunSingle('first');
		Phase	 := 3;
		Run		 := FALSE;

	3:
		IF Inner.Run(Enable := TRUE) THEN
			Phase := 4;
		END_IF

		Run := FALSE;

	4:
		Test.AssertFalse(Unknown, 'an unknown label is refused');
		Test.AssertTrue(Accepted, 'a known one is accepted');

		// It ran for real.
		ExpectedCount := 2;
		ActualCount	  := A.BodyCalls;
		Test.AssertEqual(ExpectedCount, ActualCount, 'the chosen test ran a second time');
		ExpectedCount := 1;
		ActualCount	  := B.BodyCalls;
		Test.AssertEqual(ExpectedCount, ActualCount, 'and nothing else did');

		// And recorded nothing.
		ExpectedCount := PassedBefore;
		ActualCount	  := Inner.PassedCount;
		Test.AssertEqual(ExpectedCount, ActualCount, 'the pass count did not move');
		ExpectedCount := 0;
		ActualCount	  := Inner.ErrorCount;
		Test.AssertEqual(ExpectedCount, ActualCount, 'and no error was invented');
		Run := TRUE;
END_CASE
END_METHOD

END_FUNCTION_BLOCK

// ---- Tests/Suite/TEST_SuiteWithNothingRegisteredIsComplete.TcPOU
// A project may legitimately deploy a suite with nothing registered. That is a

// clean result, not a failure - and it must be COMPLETE, or a sequencer above it

// waits forever.

//

// TestCount of zero is the signal for anyone who cares.
FUNCTION_BLOCK TEST_SuiteWithNothingRegisteredIsComplete IMPLEMENTS I_Test
VAR
	// A private suite, driven one scan per call. The outer test spans scans by

	// returning FALSE - which is the mechanism the inner suite is being asked to

	// drive, one level down.
	Inner			: TestSuite<4>;
	Budgets			: ST_TestBudgets;
	Phase			: DINT;
	Scans			: DINT;
	ExpectedCount	: UDINT;
	ActualCount		: UDINT;
	ExpectedOutcome : E_RunOutcome;
	ActualOutcome	: E_RunOutcome;
END_VAR

METHOD Run : BOOL
VAR_INPUT
	Enable : BOOL;
	Test   : I_TestAssertions;
END_VAR
Scans := Scans + 1;
IF Scans > 200 THEN
	Test.Fail('the inner suite never completed');
	Run := TRUE;
	RETURN;
END_IF

CASE Phase OF
	0:
		Inner.SetLabel('empty');
		Phase := 1;
		Run	  := FALSE;

	1:
		IF Inner.Run(Enable := TRUE) THEN
			Phase := 2;
		END_IF

		Run := FALSE;

	2:
		Test.AssertTrue(Inner.IsComplete, 'complete on the first scan');
		ExpectedCount := 0;
		ActualCount	  := Inner.TestCount;
		Test.AssertEqual(ExpectedCount, ActualCount, 'nothing registered');
		ActualCount := Inner.ErrorCount;
		Test.AssertEqual(ExpectedCount, ActualCount, 'and that is not an error');
		ExpectedOutcome := E_RunOutcome.Passed;
		ActualOutcome	:= Inner.Outcome;
		Test.AssertEqual(ExpectedOutcome, ActualOutcome, 'an empty run is not red');
		Run := TRUE;
END_CASE
END_METHOD

END_FUNCTION_BLOCK

// ---- Tests/Suite/TEST_SuiteWithNoLabelIsAFrameworkError.TcPOU
// An unnamed suite produces an unnamed node in the result document, which no CI

// system can group by. It is caught when the run starts, not silently tolerated.

//

// The tests still run - the label is a reporting problem, not a reason to refuse

// to work - but the run is marked untrustworthy.
FUNCTION_BLOCK TEST_SuiteWithNoLabelIsAFrameworkError IMPLEMENTS I_Test
VAR
	// A private suite, driven one scan per call. The outer test spans scans by

	// returning FALSE - which is the mechanism the inner suite is being asked to

	// drive, one level down.
	Inner		  : TestSuite<4>;
	Budgets		  : ST_TestBudgets;
	Phase		  : DINT;
	Scans		  : DINT;
	A			  : PassingTest;
	ExpectedCount : UDINT;
	ActualCount	  : UDINT;
END_VAR

METHOD Run : BOOL
VAR_INPUT
	Enable : BOOL;
	Test   : I_TestAssertions;
END_VAR
Scans := Scans + 1;
IF Scans > 200 THEN
	Test.Fail('the inner suite never completed');
	Run := TRUE;
	RETURN;
END_IF

CASE Phase OF
	0:
		// Deliberately no SetLabel.
		Inner.Register(A, 'a test', Budgets);
		Phase := 1;
		Run	  := FALSE;

	1:
		IF Inner.Run(Enable := TRUE) THEN
			Phase := 2;
		END_IF

		Run := FALSE;

	2:
		Test.AssertTrue(Inner.ErrorCount > 0, 'the missing label was reported');

		// The test itself still ran and still passed.
		ExpectedCount := 1;
		ActualCount	  := A.BodyCalls;
		Test.AssertEqual(ExpectedCount, ActualCount, 'the test still ran');
		ActualCount := Inner.PassedCount;
		Test.AssertEqual(ExpectedCount, ActualCount, 'and still passed');
		Run := TRUE;
END_CASE
END_METHOD

END_FUNCTION_BLOCK

// ---- Tests/Suite/TEST_SuiteDefaultsReachTheTests.TcPOU
// A suite-wide deadline reaches every test that did not claim one, and reaches it

// when the RUN starts rather than at registration - a default may be set after

// some tests are already registered.

//

// The subject hangs. With no default it would run forever and the watchdog would

// fail this test; with the default applied it times out and is reported Failed.
FUNCTION_BLOCK TEST_SuiteDefaultsReachTheTests IMPLEMENTS I_Test
VAR
	// A private suite, driven one scan per call. The outer test spans scans by

	// returning FALSE - which is the mechanism the inner suite is being asked to

	// drive, one level down.
	Inner		  : TestSuite<4>;
	Budgets		  : ST_TestBudgets;
	Phase		  : DINT;
	Scans		  : DINT;
	Hangs		  : HangingBodyTest;
	Defaults	  : ST_TestBudgets;
	ExpectedCount : UDINT;
	ActualCount	  : UDINT;
END_VAR

METHOD Run : BOOL
VAR_INPUT
	Enable : BOOL;
	Test   : I_TestAssertions;
END_VAR
Scans := Scans + 1;
IF Scans > 200 THEN
	Test.Fail('the inner suite never completed');
	Run := TRUE;
	RETURN;
END_IF

CASE Phase OF
	0:
		Inner.SetLabel('inner');

		// Registered BEFORE the default is set, which is the case that matters.
		Inner.Register(Hangs, 'hangs', Budgets);
		Defaults.Body.Cycles	  := 4;
		Defaults.Body.IsCyclesSet := TRUE;
		Inner.SetDefaults(Defaults);
		Phase := 1;
		Run	  := FALSE;

	1:
		IF Inner.Run(Enable := TRUE) THEN
			Phase := 2;
		END_IF

		Run := FALSE;

	2:
		ExpectedCount := 4;
		ActualCount	  := Hangs.BodyCalls;
		Test.AssertEqual(ExpectedCount, ActualCount, 'the default budget bounded it');
		ExpectedCount := 1;
		ActualCount	  := Inner.FailedCount;
		Test.AssertEqual(ExpectedCount, ActualCount, 'and it was reported as a failure');
		Test.AssertTrue(Inner.IsComplete, 'the suite completed rather than stalling');
		Run := TRUE;
END_CASE
END_METHOD

END_FUNCTION_BLOCK

// ---- Tests/Suite/TEST_RunAnnouncesItselfBeforeAnythingElse.TcPOU
// A run says it has begun BEFORE any result in it arrives.

//

// The ordering IS the contract, not a detail of it. A sink that opens a document

// on RunStarted has nowhere to put a result that arrived first.

//

// StartedBeforeAnything is captured by the spy at the moment RunStarted arrives, so

// this cannot pass by the calls merely having happened in some order afterwards.
FUNCTION_BLOCK TEST_RunAnnouncesItselfBeforeAnythingElse IMPLEMENTS I_Test
VAR
	Runner		  : TestRun<2>;
	Suite		  : TestSuite<2>;
	Spy			  : SpyReporter;
	Subject		  : PassingTest;
	Budgets		  : ST_TestBudgets;
	Phase		  : DINT;
	Scans		  : DINT;
	ExpectedCount : UDINT;
	ActualCount	  : UDINT;
END_VAR

METHOD Run : BOOL
VAR_INPUT
	Enable : BOOL;
	Test   : I_TestAssertions;
END_VAR
Scans := Scans + 1;
IF Scans > 200 THEN
	Test.Fail('the run never completed');
	Run := TRUE;
	RETURN;
END_IF

CASE Phase OF
	0:
		Suite.SetLabel('inner');
		Suite.Register(Subject, 'a test', Budgets);
		Runner.SetLabel('a run');
		Runner.SetTargetInfo('a target');
		Runner.AddReporter(Spy);
		Runner.AddSuite(Suite);
		Phase := 1;
		Run	  := FALSE;

	1:
		IF Runner.Run(Enable := TRUE) THEN
			Phase := 2;
		END_IF

		Run := FALSE;

	2:
		ExpectedCount := 1;
		ActualCount	  := Spy.RunStartedCalls;
		Test.AssertEqual(ExpectedCount, ActualCount, 'the run announced itself once');

		// The point of the test.
		Test.AssertTrue(Spy.StartedBeforeAnything, 'and before any test or suite result arrived');
		ActualCount := Spy.RunFinishedCalls;
		Test.AssertEqual(ExpectedCount, ActualCount, 'and finished once');

		// Both ends, so a sink can bracket what it builds.
		ActualCount := Spy.SuiteFinishedCalls;
		Test.AssertEqual(ExpectedCount, ActualCount, 'with one suite between them');
		Run := TRUE;
END_CASE
END_METHOD

END_FUNCTION_BLOCK

// ---- Tests/Suite/TEST_RunRefusingASuiteIsNeverSilent.TcPOU
// A suite refused at composition still turns the run red.
//
// THE FAILURE THIS GUARDS IS SILENT. A refused suite takes every one of its tests
// with it, so the totals simply come out smaller - and smaller totals with nothing
// failing read as a healthy run. Anyone watching pass counts sees an improvement.
//
// The refusal happens while the run is still OPEN, before the aggregate exists, so
// it has nowhere to record itself at the moment it is raised. It is held and
// re-applied when the run starts. This test is what proves the second half of that
// actually happens.
//
// A re-run re-applies it too: a suite that never made it in is still missing.
FUNCTION_BLOCK TEST_RunRefusingASuiteIsNeverSilent IMPLEMENTS I_Test
VAR
	// One slot, two suites offered.
	Runner	 : TestRun<1>;
	Accepted : TestSuite<2>;
	Refused	 : TestSuite<2>;
	Recorder : RecordingReporter;

	FirstTest  : PassingTest;
	SecondTest : PassingTest;

	Budgets : ST_TestBudgets;
	TookFirst  : BOOL;
	TookSecond : BOOL;
	Phase	: DINT;
	Scans	: DINT;

	ExpectedCount : UDINT;
	ActualCount	  : UDINT;
	ExpectedOutcome : E_RunOutcome;
	ActualOutcome	: E_RunOutcome;
END_VAR

METHOD Run : BOOL
VAR_INPUT
	Enable : BOOL;
	Test   : I_TestAssertions;
END_VAR
Scans := Scans + 1;
IF Scans > 500 THEN
	Test.Fail('the inner run never completed');
	Run := TRUE;
	RETURN;
END_IF

CASE Phase OF

0:
	Accepted.SetLabel('accepted');
	Accepted.Register(FirstTest, 'a test', Budgets);

	Refused.SetLabel('refused');
	Refused.Register(SecondTest, 'a test that will never run', Budgets);

	Runner.SetLabel('a run');
	Runner.AddReporter(Recorder);

	TookFirst  := Runner.AddSuite(Accepted);
	// One too many for a TestRun<1>.
	TookSecond := Runner.AddSuite(Refused);

	Phase := 1;
	Run	  := FALSE;

1:
	IF Runner.Run(Enable := TRUE) THEN
		Phase := 2;
	END_IF
	Run := FALSE;

2:
	Test.AssertTrue(TookFirst, 'the first suite was taken');
	Test.AssertFalse(TookSecond, 'and the second was refused');

	ExpectedCount := 1;
	ActualCount	  := Runner.SuiteCount;
	Test.AssertEqual(ExpectedCount, ActualCount, 'only one suite is in the run');

	// The whole point. The refusal happened before the aggregate existed.
	ActualCount := Runner.ErrorCount;
	Test.AssertEqual(ExpectedCount, ActualCount, 'and the refusal reached the counts');

	ExpectedOutcome := E_RunOutcome.Errored;
	ActualOutcome	:= Runner.Outcome;
	Test.AssertEqual(ExpectedOutcome, ActualOutcome, 'so the run cannot be trusted');

	// It also reached a sink, so the failure is visible without inspecting counts.
	Test.AssertTrue(Recorder.ErrorCount > 0, 'and was reported');

	// The test in the refused suite never ran - which is exactly what makes a
	// silent refusal dangerous.
	ExpectedCount := 0;
	ActualCount	  := SecondTest.BodyCalls;
	Test.AssertEqual(ExpectedCount, ActualCount, 'its tests never ran');

	Runner.ReRun();
	Phase := 3;
	Run	  := FALSE;

3:
	IF Runner.Run(Enable := TRUE) THEN
		Phase := 4;
	END_IF
	Run := FALSE;

4:
	// Still missing, so still red. A re-run must not launder a bad composition.
	ExpectedCount := 1;
	ActualCount	  := Runner.ErrorCount;
	Test.AssertEqual(ExpectedCount, ActualCount, 'the re-run is red for the same reason');

	ExpectedOutcome := E_RunOutcome.Errored;
	ActualOutcome	:= Runner.Outcome;
	Test.AssertEqual(ExpectedOutcome, ActualOutcome, 'and reports it');

	Run := TRUE;

END_CASE
END_METHOD

END_FUNCTION_BLOCK

// ---- Doubles/RecordingReporter.TcPOU
// Captures results in memory instead of writing them, so a test can ask questions

// of the ARTIFACT rather than of a counter.

//

// Every characterization test depends on it. Those tests do not ask "did a failure

// happen" - the object tests already do - they ask how many cases the document

// would carry, what type attribute a failure got, and whether a timeout message

// names the wall clock. None of that is answerable from a spy that only counts.

//

// Implements both faces. The verdicts build the case list; the detail face is

// implemented so the fan-out treats this the way it treats the JUnit writer, and

// so a test can confirm checks arrived at all.
FUNCTION_BLOCK RecordingReporter IMPLEMENTS I_TestReporter, I_TestDetailSink
VAR
	// Twenty is well past what any characterization test registers. A test that

	// overflows this is miscounting, which is why the overflow is not silent.
	_Cases			  : ARRAY[0..19] OF ST_RecordedCase;
	_CaseCount		  : UDINT;
	_SuiteCount		  : UDINT;
	_SaveCount		  : UDINT;
	_RunStartedCalls  : UDINT;
	_ErrorCount		  : UDINT;
	_LastErrorSource  : T_MaxString;
	_LastErrorText	  : T_MaxString;
	_StatTests		  : UDINT;
	_StatFailures	  : UDINT;
	_StatErrors		  : UDINT;
	_StatSkipped	  : UDINT;
	_StartedCount	  : UDINT;
	_CheckCount		  : UDINT;
	_FailedCheckCount : UDINT;
	_CasesWhenSuiteFinished : UDINT;
END_VAR

(*
	No cyclic body. Everything happens inside the notification.
*)

// The whole case at a position in arrival order, or an empty one out of range.

//

// For a test that must see what ARRIVED rather than whether a lookup succeeded:

// a label that failed to match is only diagnosable if the label is visible.
METHOD CaseAt : ST_RecordedCase
VAR_INPUT
	Index : UDINT;
END_VAR
IF Index >= _CaseCount THEN
	RETURN;
END_IF

CaseAt := _Cases[Index];
END_METHOD

// Cases recorded - the <testcase> count of the document that would be written.
PROPERTY CaseCount : UDINT
GET
CaseCount := _CaseCount;
END_GET
END_PROPERTY

METHOD CaseExists : BOOL
VAR_INPUT
	Label : T_MaxString;
END_VAR
CaseExists := (THIS^.IndexOfCase(Label) >= 0);
END_METHOD

// The failure kind recorded for this label - what the result document carries in

// its type attribute. None if the case passed or does not exist.
METHOD CaseFailureKind : E_FailureKind
VAR_INPUT
	Label : T_MaxString;
END_VAR

VAR
	Index : DINT;
END_VAR
Index := THIS^.IndexOfCase(Label);
IF Index < 0 THEN
	RETURN;
END_IF

CaseFailureKind := _Cases[Index].Kind;
END_METHOD

// The verdict recorded for this label, or NotStarted if there is no such case.
METHOD CaseStatus : E_TestStatus
VAR_INPUT
	Label : T_MaxString;
END_VAR

VAR
	Index : DINT;
END_VAR
Index := THIS^.IndexOfCase(Label);
IF Index < 0 THEN
	RETURN;
END_IF

CaseStatus := _Cases[Index].Status;
END_METHOD

// Cases recorded when the most recent SuiteFinished arrived.

//

// A document builder closes the suite element on SuiteFinished. A case arriving

// after that lands under a second suite node with no totals, so a test that cares

// about ORDER compares this with CaseCount.
PROPERTY CasesWhenSuiteFinished : UDINT
GET
CasesWhenSuiteFinished := _CasesWhenSuiteFinished;
END_GET
END_PROPERTY

PROPERTY CheckCount : UDINT
GET
CheckCount := _CheckCount;
END_GET
END_PROPERTY

METHOD CheckFailed
VAR_INPUT
	StepLabel  : T_MaxString;
	Kind	   : E_FailureKind;
	Expected   : T_MaxString;
	Actual	   : T_MaxString;
	Diagnostic : T_MaxString;
	Message	   : T_MaxString;
END_VAR
_CheckCount		  := _CheckCount + 1;
_FailedCheckCount := _FailedCheckCount + 1;
END_METHOD

METHOD CheckPassed
VAR_INPUT
	StepLabel : T_MaxString;
	Detail	  : T_MaxString;
END_VAR
_CheckCount := _CheckCount + 1;
END_METHOD

METHOD CyclicLogic
(*
	Nothing asynchronous. This sink records into memory and is done.
*)
END_METHOD

// Does the most recent framework error mention this text? Used where the old

// tests looked for an overflow case in the document - overflow is a framework

// error now, not a testcase.
METHOD ErrorContains : BOOL
VAR_INPUT
	Text : T_MaxString;
END_VAR
ErrorContains := (FIND(_LastErrorText, Text) > 0);
END_METHOD

PROPERTY ErrorCount : UDINT
GET
ErrorCount := _ErrorCount;
END_GET
END_PROPERTY

PROPERTY FailedCheckCount : UDINT
GET
FailedCheckCount := _FailedCheckCount;
END_GET
END_PROPERTY

// Does the summary recorded for this label contain this text?

//

// The characterization tests use this to check that a deadline NAMES itself -

// "after 5 cycles", "of wall time". A failure that fires for the right reason but

// says the wrong thing is still a defect: the message is what someone reads at

// three in the morning.
METHOD FailureContains : BOOL
VAR_INPUT
	Label : T_MaxString;
	Text  : T_MaxString;
END_VAR

VAR
	Index : DINT;
END_VAR
Index := THIS^.IndexOfCase(Label);
IF Index < 0 THEN
	RETURN;
END_IF

FailureContains := (FIND(_Cases[Index].Summary, Text) > 0);
END_METHOD

// Where a rejected registration, an overrunning teardown or an unwritable

// document arrives. Counted apart from cases: none of them is a test result.
METHOD FrameworkError
VAR_INPUT
	Source	: T_MaxString;
	Message : T_MaxString;
END_VAR
_ErrorCount		 := _ErrorCount + 1;
_LastErrorSource := Source;
_LastErrorText	 := Message;
END_METHOD

// Where a case with this label was recorded, or -1.

//

// Not named Find or Lookup by accident: FIND is a standard function and this

// mirrors TestRegistry.Lookup deliberately.
METHOD IndexOfCase : DINT
VAR_INPUT
	Label : T_MaxString;
END_VAR

VAR
	i : DINT;
END_VAR
IndexOfCase := -1;
IF Label = '' THEN
	RETURN;
END_IF

FOR i := 0 TO TO_DINT(_CaseCount) - 1 DO
	IF _Cases[i].Label = Label THEN
		IndexOfCase := i;
		RETURN;
	END_IF
END_FOR
END_METHOD

PROPERTY IsIdle : BOOL
GET
IsIdle := TRUE;
END_GET
END_PROPERTY

PROPERTY LastErrorSource : T_MaxString
GET
LastErrorSource := _LastErrorSource;
END_GET
END_PROPERTY

PROPERTY LastErrorText : T_MaxString
GET
LastErrorText := _LastErrorText;
END_GET
END_PROPERTY

// Back to as-declared. Called at the start of each characterization test, which

// reuses one recorder across several phases.
METHOD Reset
VAR
	i : DINT;
END_VAR
FOR i := 0 TO 19 DO
	_Cases[i].Label	   := '';
	_Cases[i].Location := '';
	_Cases[i].Summary  := '';
	_Cases[i].Status   := E_TestStatus.NotStarted;
	_Cases[i].Kind	   := E_FailureKind.None;
END_FOR

_CaseCount		 := 0;
_SuiteCount		 := 0;
_SaveCount		 := 0;
_RunStartedCalls := 0;
_ErrorCount		 := 0;
_LastErrorSource := '';
_LastErrorText	 := '';
_StatTests		 := 0;
_StatFailures	 := 0;
_StatErrors		 := 0;
_StatSkipped	 := 0;
_CasesWhenSuiteFinished := 0;
END_METHOD

// Stands in for the document being written. One run, one save - which is what

// the JUnit writer does, so counting these is counting files.
METHOD RunFinished
VAR_INPUT
	Status	   : I_TestRunStatus;
	TargetInfo : T_MaxString;
END_VAR
_SaveCount := _SaveCount + 1;
END_METHOD

METHOD RunStarted
VAR_INPUT
	Label	   : T_MaxString;
	TargetInfo : T_MaxString;
END_VAR
_RunStartedCalls := _RunStartedCalls + 1;
END_METHOD

// Documents that would have been written. One per run.
PROPERTY SaveCount : UDINT
GET
SaveCount := _SaveCount;
END_GET
END_PROPERTY

PROPERTY StartedCount : UDINT
GET
StartedCount := _StartedCount;
END_GET
END_PROPERTY

// Kept apart from StatFailures on purpose: a framework error and a failed check

// are different signals and a build should react differently to each.
PROPERTY StatErrors : UDINT
GET
StatErrors := _StatErrors;
END_GET
END_PROPERTY

PROPERTY StatFailures : UDINT
GET
StatFailures := _StatFailures;
END_GET
END_PROPERTY

PROPERTY StatSkipped : UDINT
GET
StatSkipped := _StatSkipped;
END_GET
END_PROPERTY

PROPERTY StatTests : UDINT
GET
StatTests := _StatTests;
END_GET
END_PROPERTY

// Suite nodes. Exactly one per run per suite; more than that was a real defect

// in this library history, where a reset loop appended one node per array slot.
PROPERTY SuiteCount : UDINT
GET
SuiteCount := _SuiteCount;
END_GET
END_PROPERTY

// One suite node, and the statistics it would carry.
METHOD SuiteFinished
VAR_INPUT
	Status : I_TestRunStatus;
END_VAR
IF Status = 0 THEN
	RETURN;
END_IF

_SuiteCount	  := _SuiteCount + 1;
_StatTests	  := Status.TestCount;
_StatFailures := Status.FailedCount;
_StatErrors	  := Status.ErrorCount;
_StatSkipped  := Status.SkippedCount;
_CasesWhenSuiteFinished := _CaseCount;
END_METHOD

METHOD TestFinished
VAR_INPUT
	SuiteLabel	  : T_MaxString;
	TestLabel	  : T_MaxString;
	Location	  : T_MaxString;
	Status		  : E_TestStatus;
	Kind		  : E_FailureKind;
	Summary		  : T_MaxString;
	ElapsedTime	  : LREAL;
	ElapsedCycles : UDINT;
	Assertions	  : UDINT;
END_VAR

VAR
	Index : DINT;
END_VAR
IF _CaseCount > 19 THEN
	// Silently dropping would make a miscounting test look like a passing one.
	RETURN;
END_IF

Index				   := TO_DINT(_CaseCount);
_Cases[Index].Label	   := TestLabel;
_Cases[Index].Location := Location;
_Cases[Index].Status   := Status;
_Cases[Index].Kind	   := Kind;
_Cases[Index].Summary  := Summary;
_CaseCount			   := _CaseCount + 1;
END_METHOD

METHOD TestStarted
VAR_INPUT
	SuiteLabel : T_MaxString;
	TestLabel  : T_MaxString;
	Location   : T_MaxString;
END_VAR
_StartedCount := _StartedCount + 1;
END_METHOD

END_FUNCTION_BLOCK

// ---- Tests/Suite/TEST_RunPassesWithSkipsBesideAPass.TcPOU
// A run holding a pass and some skips is Passed, whatever the number of suites.
//
// THE FAILURE THIS GUARDS IS A UNIT MISMATCH. A run folds each suite in with
// Absorb, and "all skipped" was once decided by comparing SkippedCount - a count
// of TESTS - with the number of results absorbed - a count of SUITES. Two skipped
// tests across two suites satisfied it, so a run that passed a test settled as
// Skipped, and the log sink printed it as a failed run.
//
// The shape is deliberate: two skipped tests, two suites. The collision is the
// point. TEST_RunWithMoreSkipsThanPassesIsPassed is the same run with three skips,
// which settled correctly even before the fix - the pair shows it was the
// collision, not the proportion of skips, that decided the outcome.
FUNCTION_BLOCK TEST_RunPassesWithSkipsBesideAPass IMPLEMENTS I_Test
VAR
	Runner		 : TestRun<2>;
	PassingSuite : TestSuite<2>;
	SkippedSuite : TestSuite<2>;

	Passes	   : PassingTest;
	FirstSkip  : PassingTest;
	SecondSkip : PassingTest;

	Budgets : ST_TestBudgets;
	Phase	: DINT;
	Scans	: DINT;

	ExpectedCount : UDINT;
	ActualCount	  : UDINT;
	ExpectedOutcome : E_RunOutcome;
	ActualOutcome	: E_RunOutcome;
END_VAR

METHOD Run : BOOL
VAR_INPUT
	Enable : BOOL;
	Test   : I_TestAssertions;
END_VAR
Scans := Scans + 1;
IF Scans > 200 THEN
	Test.Fail('the inner run never completed');
	Run := TRUE;
	RETURN;
END_IF

CASE Phase OF

0:
	PassingSuite.SetLabel('passing');
	PassingSuite.Register(Passes, 'a test that passes', Budgets);

	SkippedSuite.SetLabel('skipped');
	SkippedSuite.Register(FirstSkip, 'a skipped test', Budgets);
	SkippedSuite.Register(SecondSkip, 'another skipped test', Budgets);
	SkippedSuite.Skip();

	Runner.SetLabel('a run');
	Runner.AddSuite(PassingSuite);
	Runner.AddSuite(SkippedSuite);

	Phase := 1;
	Run	  := FALSE;

1:
	IF Runner.Run(Enable := TRUE) THEN
		Phase := 2;
	END_IF
	Run := FALSE;

2:
	// The counts were always right. Only what they were taken to mean was not.
	ExpectedCount := 1;
	ActualCount	  := Runner.PassedCount;
	Test.AssertEqual(ExpectedCount, ActualCount, 'one test passed');

	ExpectedCount := 2;
	ActualCount	  := Runner.SkippedCount;
	Test.AssertEqual(ExpectedCount, ActualCount, 'two were skipped');

	ActualCount := Runner.SuiteCount;
	Test.AssertEqual(ExpectedCount, ActualCount, 'across two suites - the collision this test exists for');

	ExpectedOutcome := E_RunOutcome.Passed;
	ActualOutcome	:= Runner.Outcome;
	Test.AssertEqual(ExpectedOutcome, ActualOutcome, 'a pass beside skips is Passed, not Skipped');

	Run := TRUE;

END_CASE
END_METHOD

END_FUNCTION_BLOCK

// ---- Tests/Suite/TEST_RunOfOnlySkippedTestsIsSkipped.TcPOU
// A run in which every test was skipped is Skipped - not Passed.
//
// The same defect as TEST_RunPassesWithSkipsBesideAPass, seen from the other side:
// one suite absorbed, two tests skipped, and a rule comparing the two found them
// unequal and fell through to Passed. A run that exercised nothing reported green.
//
// Skipped does not turn a build red either, so the difference is not the build's.
// It is the reader's: a rig run that skipped its integration suites should say so
// rather than claim a pass it never earned.
FUNCTION_BLOCK TEST_RunOfOnlySkippedTestsIsSkipped IMPLEMENTS I_Test
VAR
	Runner		 : TestRun<1>;
	SkippedSuite : TestSuite<2>;

	FirstSkip  : PassingTest;
	SecondSkip : PassingTest;

	Budgets : ST_TestBudgets;
	Phase	: DINT;
	Scans	: DINT;

	ExpectedCount : UDINT;
	ActualCount	  : UDINT;
	ExpectedOutcome : E_RunOutcome;
	ActualOutcome	: E_RunOutcome;
END_VAR

METHOD Run : BOOL
VAR_INPUT
	Enable : BOOL;
	Test   : I_TestAssertions;
END_VAR
Scans := Scans + 1;
IF Scans > 200 THEN
	Test.Fail('the inner run never completed');
	Run := TRUE;
	RETURN;
END_IF

CASE Phase OF

0:
	SkippedSuite.SetLabel('skipped');
	SkippedSuite.Register(FirstSkip, 'a skipped test', Budgets);
	SkippedSuite.Register(SecondSkip, 'another skipped test', Budgets);
	SkippedSuite.Skip();

	Runner.SetLabel('a run');
	Runner.AddSuite(SkippedSuite);

	Phase := 1;
	Run	  := FALSE;

1:
	IF Runner.Run(Enable := TRUE) THEN
		Phase := 2;
	END_IF
	Run := FALSE;

2:
	ExpectedCount := 2;
	ActualCount	  := Runner.SkippedCount;
	Test.AssertEqual(ExpectedCount, ActualCount, 'both tests were skipped');

	ExpectedCount := 0;
	ActualCount	  := Runner.PassedCount;
	Test.AssertEqual(ExpectedCount, ActualCount, 'and none passed');

	ExpectedOutcome := E_RunOutcome.Skipped;
	ActualOutcome	:= Runner.Outcome;
	Test.AssertEqual(ExpectedOutcome, ActualOutcome, 'a run that exercised nothing is Skipped, not Passed');

	Run := TRUE;

END_CASE
END_METHOD

END_FUNCTION_BLOCK

// ---- Tests/Suite/TEST_RunWithMoreSkipsThanPassesIsPassed.TcPOU
// A run with more skips than passes is still Passed.
//
// A CONTROL for TEST_RunPassesWithSkipsBesideAPass: the same run, with three
// skipped tests instead of two. It passed before that defect was fixed, because
// three skips across two suites never matched the suite count.
//
// Kept because the pair isolates the cause. If this one goes red, the rule has
// started weighing the proportion of skips, which would be a different defect.
FUNCTION_BLOCK TEST_RunWithMoreSkipsThanPassesIsPassed IMPLEMENTS I_Test
VAR
	Runner		 : TestRun<2>;
	PassingSuite : TestSuite<2>;
	SkippedSuite : TestSuite<4>;

	Passes	   : PassingTest;
	FirstSkip  : PassingTest;
	SecondSkip : PassingTest;
	ThirdSkip  : PassingTest;

	Budgets : ST_TestBudgets;
	Phase	: DINT;
	Scans	: DINT;

	ExpectedCount : UDINT;
	ActualCount	  : UDINT;
	ExpectedOutcome : E_RunOutcome;
	ActualOutcome	: E_RunOutcome;
END_VAR

METHOD Run : BOOL
VAR_INPUT
	Enable : BOOL;
	Test   : I_TestAssertions;
END_VAR
Scans := Scans + 1;
IF Scans > 200 THEN
	Test.Fail('the inner run never completed');
	Run := TRUE;
	RETURN;
END_IF

CASE Phase OF

0:
	PassingSuite.SetLabel('passing');
	PassingSuite.Register(Passes, 'a test that passes', Budgets);

	SkippedSuite.SetLabel('skipped');
	SkippedSuite.Register(FirstSkip, 'a skipped test', Budgets);
	SkippedSuite.Register(SecondSkip, 'another skipped test', Budgets);
	SkippedSuite.Register(ThirdSkip, 'a third skipped test', Budgets);
	SkippedSuite.Skip();

	Runner.SetLabel('a run');
	Runner.AddSuite(PassingSuite);
	Runner.AddSuite(SkippedSuite);

	Phase := 1;
	Run	  := FALSE;

1:
	IF Runner.Run(Enable := TRUE) THEN
		Phase := 2;
	END_IF
	Run := FALSE;

2:
	ExpectedCount := 1;
	ActualCount	  := Runner.PassedCount;
	Test.AssertEqual(ExpectedCount, ActualCount, 'one test passed');

	ExpectedCount := 3;
	ActualCount	  := Runner.SkippedCount;
	Test.AssertEqual(ExpectedCount, ActualCount, 'three were skipped - more than the suite count');

	ExpectedOutcome := E_RunOutcome.Passed;
	ActualOutcome	:= Runner.Outcome;
	Test.AssertEqual(ExpectedOutcome, ActualOutcome, 'more skips than passes is still Passed');

	Run := TRUE;

END_CASE
END_METHOD

END_FUNCTION_BLOCK

// ---- Tests/Suite/TEST_RunReportsASuiteSkippedBeforeItsReporters.TcPOU
// A suite skipped before any reporter was attached still reaches the reporters.
//
// Skip is only permitted before a suite is first enabled, and a composition root
// naturally skips in the block that registers - before its sinks are attached,
// and always before the run has started. Skip used to announce the suite to its
// sinks at the moment it was called, so in this order the announcement reached
// nothing: the skipped tests appeared in the run totals and in no sink at all.
//
// The wiring below is the order a consumer reported, kept as reported: register,
// skip, then label the run, attach the sink, add the suites. Skip settles the
// counts when it is called; the sinks hear about it when the run reaches the suite.
FUNCTION_BLOCK TEST_RunReportsASuiteSkippedBeforeItsReporters IMPLEMENTS I_Test
VAR
	Runner		 : TestRun<2>;
	PassingSuite : TestSuite<2>;
	SkippedSuite : TestSuite<2>;
	Spy			 : SpyReporter;

	Passes	   : PassingTest;
	FirstSkip  : PassingTest;
	SecondSkip : PassingTest;

	Budgets : ST_TestBudgets;
	Phase	: DINT;
	Scans	: DINT;

	ExpectedCount : UDINT;
	ActualCount	  : UDINT;
	ExpectedOutcome : E_RunOutcome;
	ActualOutcome	: E_RunOutcome;
END_VAR

METHOD Run : BOOL
VAR_INPUT
	Enable : BOOL;
	Test   : I_TestAssertions;
END_VAR
Scans := Scans + 1;
IF Scans > 200 THEN
	Test.Fail('the inner run never completed');
	Run := TRUE;
	RETURN;
END_IF

CASE Phase OF

0:
	PassingSuite.SetLabel('passing');
	PassingSuite.Register(Passes, 'a test that passes', Budgets);

	SkippedSuite.SetLabel('skipped');
	SkippedSuite.Register(FirstSkip, 'a skipped test', Budgets);
	SkippedSuite.Register(SecondSkip, 'another skipped test', Budgets);
	// Before any sink exists.
	SkippedSuite.Skip();

	Runner.SetLabel('a run');
	Runner.AddReporter(Spy);
	Runner.AddSuite(PassingSuite);
	Runner.AddSuite(SkippedSuite);

	Phase := 1;
	Run	  := FALSE;

1:
	IF Runner.Run(Enable := TRUE) THEN
		Phase := 2;
	END_IF
	Run := FALSE;

2:
	ExpectedCount := 2;
	ActualCount	  := Spy.SuiteFinishedCalls;
	Test.AssertEqual(ExpectedCount, ActualCount, 'both suites reached the sink, the skipped one included');

	// The skipped suite runs second, so it is the last one the sink heard about.
	ExpectedOutcome := E_RunOutcome.Skipped;
	ActualOutcome	:= Spy.LastSuiteOutcome;
	Test.AssertEqual(ExpectedOutcome, ActualOutcome, 'and it arrived as Skipped');

	Run := TRUE;

END_CASE
END_METHOD

END_FUNCTION_BLOCK

// ---- Tests/Suite/TEST_RunReportsASkippedSuiteInItsPlace.TcPOU
// A skipped suite is reported in its place in the run - after RunStarted, and
// after the suites ahead of it - not at the moment Skip was called.
//
// The companion to TEST_RunReportsASuiteSkippedBeforeItsReporters, with the sink
// attached FIRST: the order that looks as if it ought to work. It did not. Skip
// announced the suite immediately, which was before RunStarted and ahead of every
// suite that runs before it, so a sink that opens its document on RunStarted was
// handed a result for a run that, as far as it knew, had not begun.
//
// So there was no correct wiring order to document. That is why the fix moved the
// announcement instead, and why this test attaches the sink before Skip.
FUNCTION_BLOCK TEST_RunReportsASkippedSuiteInItsPlace IMPLEMENTS I_Test
VAR
	Runner		 : TestRun<2>;
	PassingSuite : TestSuite<2>;
	SkippedSuite : TestSuite<2>;
	Spy			 : SpyReporter;

	Passes	   : PassingTest;
	FirstSkip  : PassingTest;
	SecondSkip : PassingTest;

	Budgets : ST_TestBudgets;
	Phase	: DINT;
	Scans	: DINT;

	ExpectedCount : UDINT;
	ActualCount	  : UDINT;
	ExpectedOutcome : E_RunOutcome;
	ActualOutcome	: E_RunOutcome;
END_VAR

METHOD Run : BOOL
VAR_INPUT
	Enable : BOOL;
	Test   : I_TestAssertions;
END_VAR
Scans := Scans + 1;
IF Scans > 200 THEN
	Test.Fail('the inner run never completed');
	Run := TRUE;
	RETURN;
END_IF

CASE Phase OF

0:
	PassingSuite.SetLabel('passing');
	PassingSuite.Register(Passes, 'a test that passes', Budgets);

	SkippedSuite.SetLabel('skipped');
	SkippedSuite.Register(FirstSkip, 'a skipped test', Budgets);
	SkippedSuite.Register(SecondSkip, 'another skipped test', Budgets);

	// The sink reaches both suites through AddSuite before anything is skipped.
	Runner.SetLabel('a run');
	Runner.AddReporter(Spy);
	Runner.AddSuite(PassingSuite);
	Runner.AddSuite(SkippedSuite);
	SkippedSuite.Skip();

	Phase := 1;
	Run	  := FALSE;

1:
	IF Runner.Run(Enable := TRUE) THEN
		Phase := 2;
	END_IF
	Run := FALSE;

2:
	Test.AssertTrue(Spy.StartedBeforeAnything, 'the run announced itself before any suite was reported');

	ExpectedCount := 2;
	ActualCount	  := Spy.SuiteFinishedCalls;
	Test.AssertEqual(ExpectedCount, ActualCount, 'each suite was reported exactly once');

	// Reported in sequence, the skipped suite comes after the one ahead of it.
	ExpectedOutcome := E_RunOutcome.Skipped;
	ActualOutcome	:= Spy.LastSuiteOutcome;
	Test.AssertEqual(ExpectedOutcome, ActualOutcome, 'and the skipped suite was reported last, in its place');

	Run := TRUE;

END_CASE
END_METHOD

END_FUNCTION_BLOCK

// ---- Tests/Suite/TEST_RunReportsEachSkippedTestByName.TcPOU
// Every skipped test reaches the sinks by name, as a case of its own, before its
// suite is closed.
//
// The result document is what CI reads, and CI reads CASES. A suite element that
// says skipped="2" and holds no testcase children is two tests that CI cannot see,
// cannot name, and cannot trend. The JUnit writer was built to take a skipped case
// that arrives without TestStarted; nothing ever sent it one.
//
// ORDER MATTERS. A document builder closes the suite element on SuiteFinished, so a
// case that arrives after it lands under a second suite node with no totals. That
// is what CasesWhenSuiteFinished on the recorder is for.
//
// Wired in the order a consumer reported - Skip before the sink exists - so this
// also depends on the announcement having moved to when the run reaches the suite.
//
// The second skipped test has a LOCATION, and that is checked before any name. A
// skipped test never becomes active, so its journal never learns its name or its
// location; both must be taken from the registry slot. Announcing from the journal
// empties both, so if the location check fails, that is the code that ran - and
// the name checks after it print the name that actually arrived, not TRUE/FALSE.
FUNCTION_BLOCK TEST_RunReportsEachSkippedTestByName IMPLEMENTS I_Test
VAR
	Runner		 : TestRun<2>;
	PassingSuite : TestSuite<2>;
	SkippedSuite : TestSuite<2>;
	Recorder	 : RecordingReporter;

	Passes	   : PassingTest;
	FirstSkip  : PassingTest;
	// Implements I_TestLocation with a fixed path - the fingerprint above.
	SecondSkip : FakeTestWithAllHooks;

	ExpectedStatus : E_TestStatus;
	ActualStatus	: E_TestStatus;
	Recorded		: ST_RecordedCase;
	ExpectedText	: T_MaxString;
	ActualText		: T_MaxString;

	Budgets : ST_TestBudgets;
	Phase	: DINT;
	Scans	: DINT;

	ExpectedCount : UDINT;
	ActualCount	  : UDINT;
	ExpectedOutcome : E_RunOutcome;
	ActualOutcome	: E_RunOutcome;
END_VAR

METHOD Run : BOOL
VAR_INPUT
	Enable : BOOL;
	Test   : I_TestAssertions;
END_VAR
Scans := Scans + 1;
IF Scans > 200 THEN
	Test.Fail('the inner run never completed');
	Run := TRUE;
	RETURN;
END_IF

CASE Phase OF

0:
	PassingSuite.SetLabel('passing');
	PassingSuite.Register(Passes, 'a test that passes', Budgets);

	SkippedSuite.SetLabel('skipped');
	SkippedSuite.Register(FirstSkip, 'a skipped test', Budgets);
	SkippedSuite.Register(SecondSkip, 'another skipped test', Budgets);
	SkippedSuite.Skip();

	Runner.SetLabel('a run');
	Runner.AddReporter(Recorder);
	Runner.AddSuite(PassingSuite);
	Runner.AddSuite(SkippedSuite);

	Phase := 1;
	Run	  := FALSE;

1:
	IF Runner.Run(Enable := TRUE) THEN
		Phase := 2;
	END_IF
	Run := FALSE;

2:
	ExpectedCount := 3;
	ActualCount	  := Recorder.CaseCount;
	Test.AssertEqual(ExpectedCount, ActualCount, 'every test in the run is a case, the skipped two included');

	// Cases arrive in run order: the passing test, then the two skipped ones.
	Recorded	 := Recorder.CaseAt(2);
	ExpectedText := 'Verifier.Doubles.AllHooks';
	ActualText	 := Recorded.Location;
	Test.AssertEqual(ExpectedText, ActualText, 'a skipped case carries its location');

	Recorded	 := Recorder.CaseAt(1);
	ExpectedText := 'a skipped test';
	ActualText	 := Recorded.Label;
	Test.AssertEqual(ExpectedText, ActualText, 'the first skipped case arrived named');

	Recorded	 := Recorder.CaseAt(2);
	ExpectedText := 'another skipped test';
	ActualText	 := Recorded.Label;
	Test.AssertEqual(ExpectedText, ActualText, 'and so did the second');

	Test.AssertTrue(Recorder.CaseExists('a skipped test'), 'the first skipped test is there by name');
	ExpectedStatus := E_TestStatus.Skipped;
	ActualStatus	:= Recorder.CaseStatus('a skipped test');
	Test.AssertEqual(ExpectedStatus, ActualStatus, 'and recorded as Skipped');

	Test.AssertTrue(Recorder.CaseExists('another skipped test'), 'so is the second');
	ActualStatus := Recorder.CaseStatus('another skipped test');
	Test.AssertEqual(ExpectedStatus, ActualStatus, 'also as Skipped');

	// All three cases had arrived when the last suite - the skipped one - closed.
	ActualCount := Recorder.CasesWhenSuiteFinished;
	Test.AssertEqual(ExpectedCount, ActualCount, 'the skipped cases arrived before their suite was closed');

	ExpectedCount := 2;
	ActualCount	  := Recorder.SuiteCount;
	Test.AssertEqual(ExpectedCount, ActualCount, 'and each suite was closed exactly once');

	Run := TRUE;

END_CASE
END_METHOD

END_FUNCTION_BLOCK

// ---- Tests/Suite/TEST_RunReRunDoesNotRunASkippedSuite.TcPOU
// A re-run does not run the tests of a skipped suite. They stay skipped.
//
// THE HAZARD. A suite is skipped because running it would be wrong here - the
// hardware is absent, or present and not to be moved. A run-level ReRun once
// re-executed every suite's registered tests, skipped or not, so the one button
// meant for someone at a keyboard ran exactly the tests that had been ruled out.
//
// Skip is part of composition, and a re-run "re-executes what was composed; it
// does not recompose it" (TestRun.ReRun). A skip is part of what was composed.
//
// The passing test must run TWICE. Without that, a re-run that silently did
// nothing would pass every other check here.
FUNCTION_BLOCK TEST_RunReRunDoesNotRunASkippedSuite IMPLEMENTS I_Test
VAR
	Runner		 : TestRun<2>;
	PassingSuite : TestSuite<2>;
	SkippedSuite : TestSuite<2>;

	Passes	   : PassingTest;
	FirstSkip  : PassingTest;
	SecondSkip : PassingTest;

	Budgets : ST_TestBudgets;
	Phase	: DINT;
	Scans	: DINT;

	ExpectedCount : UDINT;
	ActualCount	  : UDINT;
	ExpectedOutcome : E_RunOutcome;
	ActualOutcome	: E_RunOutcome;
END_VAR

METHOD Run : BOOL
VAR_INPUT
	Enable : BOOL;
	Test   : I_TestAssertions;
END_VAR
Scans := Scans + 1;
IF Scans > 200 THEN
	Test.Fail('the inner run never completed');
	Run := TRUE;
	RETURN;
END_IF

CASE Phase OF

0:
	PassingSuite.SetLabel('passing');
	PassingSuite.Register(Passes, 'a test that passes', Budgets);

	SkippedSuite.SetLabel('skipped');
	SkippedSuite.Register(FirstSkip, 'a skipped test', Budgets);
	SkippedSuite.Register(SecondSkip, 'another skipped test', Budgets);
	SkippedSuite.Skip();

	Runner.SetLabel('a run');
	Runner.AddSuite(PassingSuite);
	Runner.AddSuite(SkippedSuite);

	Phase := 1;
	Run	  := FALSE;

1:
	IF Runner.Run(Enable := TRUE) THEN
		Phase := 2;
	END_IF
	Run := FALSE;

2:
	// The house way to re-run: once the first pass is complete.
	Runner.ReRun();
	Phase := 3;
	Run	  := FALSE;

3:
	IF Runner.Run(Enable := TRUE) THEN
		Phase := 4;
	END_IF
	Run := FALSE;

4:
	ExpectedCount := 2;
	ActualCount	  := Passes.BodyCalls;
	Test.AssertEqual(ExpectedCount, ActualCount, 'the re-run really ran: the passing test ran twice');

	ExpectedCount := 0;
	ActualCount	  := FirstSkip.BodyCalls;
	Test.AssertEqual(ExpectedCount, ActualCount, 'a skipped test never ran, not even in the re-run');
	ActualCount := SecondSkip.BodyCalls;
	Test.AssertEqual(ExpectedCount, ActualCount, 'nor did the other');

	ExpectedCount := 2;
	ActualCount	  := Runner.SkippedCount;
	Test.AssertEqual(ExpectedCount, ActualCount, 'the re-run still counts them skipped');
	ExpectedCount := 1;
	ActualCount	  := Runner.PassedCount;
	Test.AssertEqual(ExpectedCount, ActualCount, 'and counts the one pass once, not twice');

	Run := TRUE;

END_CASE
END_METHOD

END_FUNCTION_BLOCK

// ---- Tests/Suite/TEST_RunReRunReportsASkippedSuiteAgain.TcPOU
// A re-run reports a skipped suite again - its tests by name, then the suite -
// and reports it as Skipped.
//
// A re-run exists to produce a FRESH document. If the skipped suite said nothing
// the second time, its tests would vanish from that document; if its tests ran,
// they would appear as passes that were never meant to happen. Either way the
// re-run's artifact would disagree with the first run's about what was skipped.
//
// The skipped suite is added last, so what the sink heard LAST is its report.
FUNCTION_BLOCK TEST_RunReRunReportsASkippedSuiteAgain IMPLEMENTS I_Test
VAR
	Runner		 : TestRun<2>;
	PassingSuite : TestSuite<2>;
	SkippedSuite : TestSuite<2>;
	Spy			 : SpyReporter;

	Passes	   : PassingTest;
	FirstSkip  : PassingTest;
	SecondSkip : PassingTest;

	Budgets : ST_TestBudgets;
	Phase	: DINT;
	Scans	: DINT;

	ExpectedCount : UDINT;
	ActualCount	  : UDINT;
	ExpectedOutcome : E_RunOutcome;
	ActualOutcome	: E_RunOutcome;
	ExpectedStatus : E_TestStatus;
	ActualStatus	: E_TestStatus;
END_VAR

METHOD Run : BOOL
VAR_INPUT
	Enable : BOOL;
	Test   : I_TestAssertions;
END_VAR
Scans := Scans + 1;
IF Scans > 200 THEN
	Test.Fail('the inner run never completed');
	Run := TRUE;
	RETURN;
END_IF

CASE Phase OF

0:
	PassingSuite.SetLabel('passing');
	PassingSuite.Register(Passes, 'a test that passes', Budgets);

	SkippedSuite.SetLabel('skipped');
	SkippedSuite.Register(FirstSkip, 'a skipped test', Budgets);
	SkippedSuite.Register(SecondSkip, 'another skipped test', Budgets);
	SkippedSuite.Skip();

	Runner.SetLabel('a run');
	Runner.AddReporter(Spy);
	Runner.AddSuite(PassingSuite);
	Runner.AddSuite(SkippedSuite);

	Phase := 1;
	Run	  := FALSE;

1:
	IF Runner.Run(Enable := TRUE) THEN
		Phase := 2;
	END_IF
	Run := FALSE;

2:
	// The house way to re-run: once the first pass is complete.
	Runner.ReRun();
	Phase := 3;
	Run	  := FALSE;

3:
	IF Runner.Run(Enable := TRUE) THEN
		Phase := 4;
	END_IF
	Run := FALSE;

4:
	ExpectedCount := 2;
	ActualCount	  := Spy.RunFinishedCalls;
	Test.AssertEqual(ExpectedCount, ActualCount, 'the re-run finished, so a fresh document was written');

	ExpectedCount := 4;
	ActualCount	  := Spy.SuiteFinishedCalls;
	Test.AssertEqual(ExpectedCount, ActualCount, 'each suite was reported once per pass');
	ExpectedCount := 6;
	ActualCount	  := Spy.TestFinishedCalls;
	Test.AssertEqual(ExpectedCount, ActualCount, 'and each test once per pass, the skipped ones included');

	ExpectedOutcome := E_RunOutcome.Skipped;
	ActualOutcome	:= Spy.LastSuiteOutcome;
	Test.AssertEqual(ExpectedOutcome, ActualOutcome, 'the re-run reported the skipped suite as Skipped');

	ExpectedStatus := E_TestStatus.Skipped;
	ActualStatus	:= Spy.LastStatus;
	Test.AssertEqual(ExpectedStatus, ActualStatus, 'and its tests as Skipped, not as passes');

	Run := TRUE;

END_CASE
END_METHOD

END_FUNCTION_BLOCK

// ---- Tests/Fanout/TEST_FanoutNotifiesEverySinkInOrder.TcPOU
// Every attached sink receives everything, in the order it was attached.

//

// Order matters for one thing only: it is what a build can rely on if two sinks

// must not be interleaved. If sequencing between two sinks matters beyond that,

// that is one sink wrapping two - not something the fan-out should arbitrate.
FUNCTION_BLOCK TEST_FanoutNotifiesEverySinkInOrder IMPLEMENTS I_Test
VAR
	Fanout		  : TestReporterFanout;
	SpyOne		  : SpyReporter;
	SpyTwo		  : SpyReporter;
	SpyThree	  : SpyReporter;
	Witness		  : OrderWitness;
	AttachedAll	  : BOOL;
	ExpectedCount : UDINT;
	ActualCount	  : UDINT;
	ExpectedOrder : T_MaxString;
	ActualOrder	  : T_MaxString;
END_VAR

METHOD Run : BOOL
VAR_INPUT
	Enable : BOOL;
	Test   : I_TestAssertions;
END_VAR
SpyOne.Configure(1, Witness);
SpyTwo.Configure(2, Witness);
SpyThree.Configure(3, Witness);
AttachedAll := Fanout.Attach(SpyOne) AND Fanout.Attach(SpyTwo) AND Fanout.Attach(SpyThree);
Test.AssertTrue(AttachedAll, 'all three attached');
ExpectedCount := 3;
ActualCount	  := Fanout.Count;
Test.AssertEqual(ExpectedCount, ActualCount, 'and Count says so');
Fanout.TestFinished(SuiteLabel	  := 'suite',
					TestLabel	  := 'a test',
					Location	  := '',
					Status		  := E_TestStatus.Passed,
					Kind		  := E_FailureKind.None,
					Summary		  := '',
					ElapsedTime	  := 0.0,
					ElapsedCycles := 0,
					Assertions	  := 1);

ExpectedCount := 1;
ActualCount	  := SpyOne.TestFinishedCalls;
Test.AssertEqual(ExpectedCount, ActualCount, 'the first was told');
ActualCount := SpyThree.TestFinishedCalls;
Test.AssertEqual(ExpectedCount, ActualCount, 'and so was the last');
ExpectedOrder := '1,2,3';
ActualOrder	  := Witness.Sequence;
Test.AssertEqual(ExpectedOrder, ActualOrder, 'in the order they were attached');

// Cyclic work reaches everyone too, and is what lets a slow sink finish.
Fanout.CyclicLogic();
ActualCount := SpyTwo.CyclicCalls;
Test.AssertEqual(ExpectedCount, ActualCount, 'and CyclicLogic reaches them all');
Run := TRUE;
END_METHOD

END_FUNCTION_BLOCK

// ---- Doubles/OrderWitness.TcPOU
// Records the order spies were notified in, as a string like '1,2,3'.

//

// A string rather than an array because the assertion reads better and because the

// whole point is to compare against a literal the reader can see.
FUNCTION_BLOCK OrderWitness IMPLEMENTS I_ProbeWitness
VAR
	_Sequence : T_MaxString;
	_Count	  : UDINT;
END_VAR

METHOD Clear
_Sequence := '';
_Count	  := 0;
END_METHOD

METHOD Note
VAR_INPUT
	Ordinal : UDINT;
END_VAR
IF _Count > 0 THEN
	_Sequence := CONCAT(_Sequence, ',');
END_IF

_Sequence := CONCAT(_Sequence, UDINT_TO_STRING(Ordinal));
_Count	  := _Count + 1;
END_METHOD

// The ordinals in the order they arrived, comma separated.
PROPERTY Sequence : T_MaxString
GET
Sequence := _Sequence;
END_GET
END_PROPERTY

END_FUNCTION_BLOCK

// ---- Tests/Fanout/TEST_FanoutOnlyChecksGoToDetailSinks.TcPOU
// A reporter that only wants verdicts is never called for a check, and does not

// write empty method bodies to say so.

//

// The fan-out asks ONCE, when the sink is attached, and remembers. A per-check

// __QUERYINTERFACE would put an interface lookup in the hottest path in the

// library - a forty-check test would pay for forty of them.
FUNCTION_BLOCK TEST_FanoutOnlyChecksGoToDetailSinks IMPLEMENTS I_Test
VAR
	Fanout		  : TestReporterFanout;
	Detailed	  : SpyReporter;
	VerdictOnly	  : VerdictOnlyReporter;
	ExpectedCount : UDINT;
	ActualCount	  : UDINT;
END_VAR

METHOD Run : BOOL
VAR_INPUT
	Enable : BOOL;
	Test   : I_TestAssertions;
END_VAR
Fanout.Attach(Detailed);
Fanout.Attach(VerdictOnly);
Fanout.TestStarted(SuiteLabel := 'suite', TestLabel := 'a test', Location := '');
Fanout.CheckPassed(StepLabel := '', Detail := '');
Fanout.CheckFailed(StepLabel  := '',
				   Kind		  := E_FailureKind.ValueMismatch,
				   Expected	  := '1',
				   Actual	  := '2',
				   Diagnostic := 'expected 1, actual 2',
				   Message	  := 'deliberate');

ExpectedCount := 1;
ActualCount	  := Detailed.TestStartedCalls;
Test.AssertEqual(ExpectedCount, ActualCount, 'the detail sink was opened');
ExpectedCount := 2;
ActualCount	  := Detailed.CheckCalls;
Test.AssertEqual(ExpectedCount, ActualCount, 'and got both checks');

// The values arrive in their own fields, not buried in the diagnostic.
Test.AssertTrue(Detailed.LastExpected = '1', 'expected travelled in its own field');
Test.AssertTrue(Detailed.LastActual = '2', 'and so did actual');

// The verdict-only sink still gets verdicts.
Fanout.TestFinished(SuiteLabel	  := 'suite',
					TestLabel	  := 'a test',
					Location	  := '',
					Status		  := E_TestStatus.Passed,
					Kind		  := E_FailureKind.None,
					Summary		  := '',
					ElapsedTime	  := 0.0,
					ElapsedCycles := 0,
					Assertions	  := 1);

ExpectedCount := 1;
ActualCount	  := VerdictOnly.TestFinishedCalls;
Test.AssertEqual(ExpectedCount, ActualCount, 'the verdict-only sink got the verdict');
Run := TRUE;
END_METHOD

END_FUNCTION_BLOCK

// ---- Doubles/VerdictOnlyReporter.TcPOU
// A reporter that wants verdicts and NOT individual checks - the event logger and

// the alarm block are both this shape.

//

// It implements I_TestReporter and deliberately not I_TestDetailSink, which is the

// whole point: it should never be called for a check, and it should not have to

// write empty method bodies to say so. The fan-out asks once, when it is attached,

// and remembers the answer.
FUNCTION_BLOCK VerdictOnlyReporter IMPLEMENTS I_TestReporter
VAR
	_CyclicCalls		 : UDINT;
	_TestFinishedCalls	 : UDINT;
	_SuiteFinishedCalls	 : UDINT;
	_RunFinishedCalls	 : UDINT;
	_RunStartedCalls	 : UDINT;
	_FrameworkErrorCalls : UDINT;
END_VAR

PROPERTY CyclicCalls : UDINT
GET
CyclicCalls := _CyclicCalls;
END_GET
END_PROPERTY

METHOD CyclicLogic
_CyclicCalls := _CyclicCalls + 1;
END_METHOD

METHOD FrameworkError
VAR_INPUT
	Source	: T_MaxString;
	Message : T_MaxString;
END_VAR
_FrameworkErrorCalls := _FrameworkErrorCalls + 1;
END_METHOD

PROPERTY FrameworkErrorCalls : UDINT
GET
FrameworkErrorCalls := _FrameworkErrorCalls;
END_GET
END_PROPERTY

PROPERTY IsIdle : BOOL
GET
IsIdle := TRUE;
END_GET
END_PROPERTY

METHOD RunFinished
VAR_INPUT
	Status	   : I_TestRunStatus;
	TargetInfo : T_MaxString;
END_VAR
_RunFinishedCalls := _RunFinishedCalls + 1;
END_METHOD

PROPERTY RunFinishedCalls : UDINT
GET
RunFinishedCalls := _RunFinishedCalls;
END_GET
END_PROPERTY

METHOD RunStarted
VAR_INPUT
	Label	   : T_MaxString;
	TargetInfo : T_MaxString;
END_VAR
_RunStartedCalls := _RunStartedCalls + 1;
END_METHOD

METHOD SuiteFinished
VAR_INPUT
	Status : I_TestRunStatus;
END_VAR
_SuiteFinishedCalls := _SuiteFinishedCalls + 1;
END_METHOD

PROPERTY SuiteFinishedCalls : UDINT
GET
SuiteFinishedCalls := _SuiteFinishedCalls;
END_GET
END_PROPERTY

METHOD TestFinished
VAR_INPUT
	SuiteLabel	  : T_MaxString;
	TestLabel	  : T_MaxString;
	Location	  : T_MaxString;
	Status		  : E_TestStatus;
	Kind		  : E_FailureKind;
	Summary		  : T_MaxString;
	ElapsedTime	  : LREAL;
	ElapsedCycles : UDINT;
	Assertions	  : UDINT;
END_VAR
_TestFinishedCalls := _TestFinishedCalls + 1;
END_METHOD

PROPERTY TestFinishedCalls : UDINT
GET
TestFinishedCalls := _TestFinishedCalls;
END_GET
END_PROPERTY

END_FUNCTION_BLOCK

// ---- Tests/Fanout/TEST_FanoutIsIdleIsTheAndOfEverySink.TcPOU
// CI must wait for IsIdle as well as IsComplete. A run finishing and its result

// document reaching disk are different events, and copying between them yields a

// truncated artifact - which reads as a broken pipeline rather than a finished run.

//

// One busy sink is enough to hold the whole fan-out busy.
FUNCTION_BLOCK TEST_FanoutIsIdleIsTheAndOfEverySink IMPLEMENTS I_Test
VAR
	Fanout : TestReporterFanout;
	Quick  : SpyReporter;
	Slow   : SpyReporter;
	Empty  : TestReporterFanout;
END_VAR

METHOD Run : BOOL
VAR_INPUT
	Enable : BOOL;
	Test   : I_TestAssertions;
END_VAR
// Nothing attached: no sink, no pending work.
Test.AssertTrue(Empty.IsIdle, 'an empty fan-out is idle');
Fanout.Attach(Quick);
Fanout.Attach(Slow);
Test.AssertTrue(Fanout.IsIdle, 'idle while both sinks are');
Slow.SetBusy(TRUE);
Test.AssertFalse(Fanout.IsIdle, 'one busy sink holds the whole fan-out busy');

// CyclicLogic is what lets a slow sink finish, so it must keep running.
Fanout.CyclicLogic();
Test.AssertTrue(Slow.CyclicCalls > 0, 'and the busy sink still gets advanced');
Slow.SetBusy(FALSE);
Test.AssertTrue(Fanout.IsIdle, 'idle again once it finishes');
Run := TRUE;
END_METHOD

END_FUNCTION_BLOCK

// ---- Tests/Fanout/TEST_FanoutSuspendSilencesEverything.TcPOU
// Suspending is how an individual re-run records nothing and saves nothing: the

// suite silences every sink at once, rather than a condition threaded through the

// runner and the journal and remembered in three places.

//

// CyclicLogic is NOT suppressed. A file write already in flight must still finish,

// or IsIdle never goes TRUE and CI waits forever.
FUNCTION_BLOCK TEST_FanoutSuspendSilencesEverything IMPLEMENTS I_Test
VAR
	Fanout		  : TestReporterFanout;
	Spy			  : SpyReporter;
	ExpectedCount : UDINT;
	ActualCount	  : UDINT;
END_VAR

METHOD Run : BOOL
VAR_INPUT
	Enable : BOOL;
	Test   : I_TestAssertions;
END_VAR
Fanout.Attach(Spy);
Fanout.Suspend();
Fanout.TestFinished(SuiteLabel	  := '',
					TestLabel	  := 'ignored',
					Location	  := '',
					Status		  := E_TestStatus.Passed,
					Kind		  := E_FailureKind.None,
					Summary		  := '',
					ElapsedTime	  := 0.0,
					ElapsedCycles := 0,
					Assertions	  := 0);

Fanout.FrameworkError(Source := '', Message := 'ignored');
Fanout.TestStarted(SuiteLabel := '', TestLabel := 'ignored', Location := '');
Fanout.CheckPassed(StepLabel := '', Detail := '');
ExpectedCount := 0;
ActualCount	  := Spy.TestFinishedCalls;
Test.AssertEqual(ExpectedCount, ActualCount, 'no verdict reached the sink');
ActualCount := Spy.FrameworkErrorCalls;
Test.AssertEqual(ExpectedCount, ActualCount, 'nor a framework error');
ActualCount := Spy.CheckCalls;
Test.AssertEqual(ExpectedCount, ActualCount, 'nor a check');

// Work in flight must still be advanced.
Fanout.CyclicLogic();
Test.AssertTrue(Spy.CyclicCalls > 0, 'but CyclicLogic is not suppressed');
Fanout.Resume();
Fanout.TestFinished(SuiteLabel	  := '',
					TestLabel	  := 'counted',
					Location	  := '',
					Status		  := E_TestStatus.Passed,
					Kind		  := E_FailureKind.None,
					Summary		  := '',
					ElapsedTime	  := 0.0,
					ElapsedCycles := 0,
					Assertions	  := 0);

ExpectedCount := 1;
ActualCount	  := Spy.TestFinishedCalls;
Test.AssertEqual(ExpectedCount, ActualCount, 'and notifications resume');

// Nothing is replayed - it was deliberately not recorded.
Test.AssertTrue(Spy.LastTestLabel = 'counted', 'the suspended one was not replayed');
Run := TRUE;
END_METHOD

END_FUNCTION_BLOCK

// ---- Tests/Fanout/TEST_FanoutRefusesBeyondCapacityAndTellsTheRest.TcPOU
// A refused attachment is reported through the sinks ALREADY attached. That reads

// circular and is not: the ones already there are exactly the ones that can still

// report it.

//

// A rejection with nothing attached at all is genuinely silent, which is why Count

// exists - assert it in CI. A sink that stops being attached takes its output with

// it, and a result file that never appears reads as a broken build rather than a

// missing sink.
FUNCTION_BLOCK TEST_FanoutRefusesBeyondCapacityAndTellsTheRest IMPLEMENTS I_Test
VAR
	Fanout		  : TestReporterFanout;
	Spies		  : ARRAY[0..8] OF SpyReporter;
	NoSink		  : I_TestReporter;
	i			  : DINT;
	Accepted	  : BOOL;
	Refused		  : BOOL;
	RefusedNull	  : BOOL;
	ExpectedCount : UDINT;
	ActualCount	  : UDINT;
END_VAR

METHOD Run : BOOL
VAR_INPUT
	Enable : BOOL;
	Test   : I_TestAssertions;
END_VAR
// Fill it to the parameter capacity, whatever that is set to.
FOR i := 0 TO TO_DINT(TestHarnessParameter.ReporterCapacity) - 1 DO
	Accepted := Fanout.Attach(Spies[i]);
	Test.AssertTrue(Accepted, 'accepted up to capacity');
END_FOR

ExpectedCount := TestHarnessParameter.ReporterCapacity;
ActualCount	  := Fanout.Count;
Test.AssertEqual(ExpectedCount, ActualCount, 'Count matches capacity');
Refused := Fanout.Attach(Spies[8]);
Test.AssertFalse(Refused, 'one beyond capacity is refused');
ActualCount := Fanout.Count;
Test.AssertEqual(ExpectedCount, ActualCount, 'and took no slot');

// Reported through the sinks that were already there.
Test.AssertTrue(Spies[0].FrameworkErrorCalls > 0, 'the refusal was reported');
RefusedNull := Fanout.Attach(NoSink);
Test.AssertFalse(RefusedNull, 'a null reporter is refused too');
Run := TRUE;
END_METHOD

END_FUNCTION_BLOCK

// ---- Tests/Fanout/TEST_FanoutCarriesTheSuiteResultThrough.TcPOU
// SuiteFinished hands the sink the read model, not a copy of the numbers. A sink

// asking a live I_TestRunStatus is what lets a JUnit writer emit counts it did not

// have to be told.
FUNCTION_BLOCK TEST_FanoutCarriesTheSuiteResultThrough IMPLEMENTS I_Test
VAR
	Fanout			: TestReporterFanout;
	Spy				: SpyReporter;
	Tally			: TestRunTally;
	ExpectedCount	: UDINT;
	ActualCount		: UDINT;
	ExpectedOutcome : E_RunOutcome;
	ActualOutcome	: E_RunOutcome;
END_VAR

METHOD Run : BOOL
VAR_INPUT
	Enable : BOOL;
	Test   : I_TestAssertions;
END_VAR
Fanout.Attach(Spy);
Tally.SetLabel('a suite');
Tally.Begin(2);
Tally.Record(Verdict := E_TestStatus.Passed, ElapsedTime := 0.1);
Tally.Record(Verdict := E_TestStatus.Failed, ElapsedTime := 0.2);
Tally.Finish();
Fanout.SuiteFinished(Tally);
ExpectedCount := 1;
ActualCount	  := Spy.SuiteFinishedCalls;
Test.AssertEqual(ExpectedCount, ActualCount, 'the sink was told once');

// Read back THROUGH the interface the sink was handed.
ActualCount := Spy.LastSuitePassed;
Test.AssertEqual(ExpectedCount, ActualCount, 'and could read the counts');
ExpectedOutcome := E_RunOutcome.Failed;
ActualOutcome	:= Spy.LastSuiteOutcome;
Test.AssertEqual(ExpectedOutcome, ActualOutcome, 'and the outcome');
Run := TRUE;
END_METHOD

END_FUNCTION_BLOCK

// ---- Tests/Fanout/TEST_FanoutForwardsRunStarted.TcPOU
// RunStarted reaches every sink, and is silenced by Suspend like any other

// notification.

//

// It is the counterpart of I_TestDetailSink.TestStarted: a sink that BUILDS

// something needs telling when to open it, rather than inferring it from the first

// thing that happens to arrive.
FUNCTION_BLOCK TEST_FanoutForwardsRunStarted IMPLEMENTS I_Test
VAR
	Fanout		  : TestReporterFanout;
	SpyOne		  : SpyReporter;
	SpyTwo		  : SpyReporter;
	ExpectedCount : UDINT;
	ActualCount	  : UDINT;
END_VAR

METHOD Run : BOOL
VAR_INPUT
	Enable : BOOL;
	Test   : I_TestAssertions;
END_VAR
Fanout.Attach(SpyOne);
Fanout.Attach(SpyTwo);
Fanout.RunStarted(Label := 'a run', TargetInfo := 'a target');
ExpectedCount := 1;
ActualCount	  := SpyOne.RunStartedCalls;
Test.AssertEqual(ExpectedCount, ActualCount, 'the first sink was told');
ActualCount := SpyTwo.RunStartedCalls;
Test.AssertEqual(ExpectedCount, ActualCount, 'and so was the second');

// Suspended, as an individual re-run does.
Fanout.Suspend();
Fanout.RunStarted(Label := 'ignored', TargetInfo := '');
ActualCount := SpyOne.RunStartedCalls;
Test.AssertEqual(ExpectedCount, ActualCount, 'and Suspend silences it too');
Run := TRUE;
END_METHOD

END_FUNCTION_BLOCK

// ---- Tests/LogReporter/TEST_LogReporterIsQuietAboutPasses.TcPOU
// Quiet by default. Eighty green lines hide the two that matter, and the counts

// are already available through I_TestRunStatus for anyone who wants them.//

// WHAT THIS CANNOT CHECK: whether the line actually reached the TwinCAT log, or

// what it says. ADSLOGSTR gives no answer back. The counters prove which BRANCH

// was taken; the wording has to be read once, by eye, in the Logged Events window.

// Saying so is better than a test that implies more than it establishes.
FUNCTION_BLOCK TEST_LogReporterIsQuietAboutPasses IMPLEMENTS I_Test
VAR
	Sink		  : TestLogReporter;
	ExpectedCount : UDINT;
	ActualCount	  : UDINT;
END_VAR

METHOD Run : BOOL
VAR_INPUT
	Enable : BOOL;
	Test   : I_TestAssertions;
END_VAR
Sink.TestFinished(SuiteLabel	:= 'suite',
				  TestLabel		:= 'a pass',
				  Location		:= '',
				  Status		:= E_TestStatus.Passed,
				  Kind			:= E_FailureKind.None,
				  Summary		:= '',
				  ElapsedTime	:= 0.0,
				  ElapsedCycles := 1,
				  Assertions	:= 1);

Sink.TestFinished(SuiteLabel	:= 'suite',
				  TestLabel		:= 'a skip',
				  Location		:= '',
				  Status		:= E_TestStatus.Skipped,
				  Kind			:= E_FailureKind.None,
				  Summary		:= '',
				  ElapsedTime	:= 0.0,
				  ElapsedCycles := 0,
				  Assertions	:= 0);

